KUKA KRL program: MyProgram_032().src

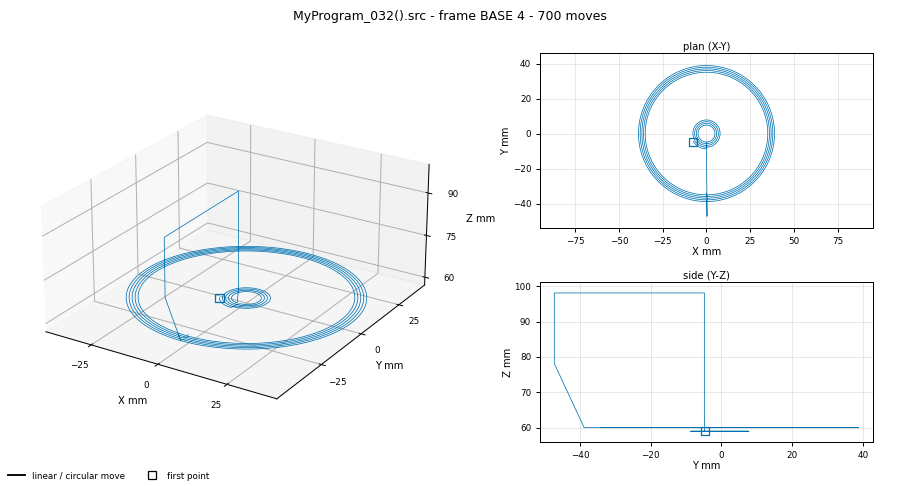
[picture p0: tool path of MyProgram_032().src in frame BASE 4, 700 of 700 moves have a stored position in this frame; points joined in program order, loops and branches not executed]
&ACCESS RVP
&REL 1
&PARAM TEMPLATE = C:\KRC\Roboter\Template\vorgabe
&PARAM EDITMASK = *
DEF MyProgram_032()
; ---- Setting reference (Base) ----
$BASE = BASE_DATA[4]

; --------------------------
; ---- Setting tool (TCP) ----
$TOOL = TOOL_DATA[3]
; --------------------------

$VEL.CP = VEL_APROX_PRINT
Startdeposition()
$VEL.CP = VEL_PRINT
LIN {X -7.455,Y -4.6001,Z 59,A -2.6784,B 0.0017,C -0.0013,E1 0.1616,E2 -630.3527} C_DIS
LIN {X -6.8252,Y -5.4917,Z 59,A -2.6167,B 0.0016,C -0.0015,E1 0.1614,E2 -630.4294} C_DIS
LIN {X -6.0357,Y -6.3443,Z 59,A -2.5577,B 0.0014,C -0.0017,E1 0.1613,E2 -630.4962} C_DIS
LIN {X -5.4394,Y -6.8632,Z 59,A -2.5125,B 0.0012,C -0.0017,E1 0.1611,E2 -630.5421} C_DIS
LIN {X -4.4516,Y -7.5448,Z 59,A -2.4498,B 0.001,C -0.0019,E1 0.1609,E2 -630.5983} C_DIS
LIN {X -3.5499,Y -8.0085,Z 59,A -2.3908,B 0.0007,C -0.002,E1 0.1606,E2 -630.6447} C_DIS
LIN {X -2.4797,Y -8.4018,Z 59,A -2.3387,B 0.0005,C -0.0021,E1 0.1604,E2 -630.6751} C_DIS
LIN {X -1.4775,Y -8.6348,Z 59,A -2.2933,B 0.0002,C -0.0021,E1 0.1601,E2 -630.6944} C_DIS
LIN {X -0.6022,Y -8.7394,Z 59,A -2.2586,B 0,C -0.0021,E1 0.1599,E2 -630.702} C_DIS
LIN {X -0.6022,Y -8.7394,Z 59,A -2.2586,B 0,C -0.0021,E1 0.1599,E2 -630.702} C_DIS
Enddeposition()
LIN {X -0.0216,Y -7.7786,Z 59,A -2.2094,B 0,C -0.0021,E1 0.1599,E2 -630.6884} C_DIS
Startdeposition()
$VEL.CP = VEL_PRINT
LIN {X -1.2171,Y -7.6837,Z 59,A -2.2663,B 0.0003,C -0.0021,E1 0.1602,E2 -630.6706} C_DIS
LIN {X -2.1503,Y -7.4764,Z 59,A -2.3206,B 0.0006,C -0.0021,E1 0.1605,E2 -630.641} C_DIS
LIN {X -3.7783,Y -6.8003,Z 59,A -2.4144,B 0.001,C -0.0019,E1 0.1609,E2 -630.5769} C_DIS
LIN {X -4.6899,Y -6.2006,Z 59,A -2.4825,B 0.0013,C -0.0017,E1 0.1611,E2 -630.5161} C_DIS
LIN {X -5.3546,Y -5.6349,Z 59,A -2.5373,B 0.0014,C -0.0016,E1 0.1613,E2 -630.4612} C_DIS
LIN {X -5.9536,Y -5,Z 59,A -2.5956,B 0.0016,C -0.0014,E1 0.1615,E2 -630.3975} C_DIS
LIN {X -6.5989,Y -4.12,Z 59,A -2.6888,B 0.0018,C -0.0011,E1 0.1617,E2 -630.2903} C_DIS
LIN {X -7.3187,Y -2.6373,Z 59,A -2.7822,B 0.002,C -0.0007,E1 0.1618,E2 -630.1603} C_DIS
LIN {X -7.6546,Y -1.3881,Z 59,A -2.8749,B 0.002,C -0.0004,E1 0.1618,E2 -630.0272} C_DIS
LIN {X -7.776,Y -0.1143,Z 59,A -2.9313,B 0.0021,C -0.0001,E1 0.1619,E2 -629.9218} C_DIS
LIN {X -7.7529,Y 0.5778,Z 59,A -2.9623,B 0.0021,C 0.0001,E1 0.1619,E2 -629.8608} C_DIS
LIN {X -7.6134,Y 1.5989,Z 59,A -3.0373,B 0.0021,C 0.0004,E1 0.1619,E2 -629.7382} C_DIS
LIN {X -7.182,Y 2.9893,Z 59,A -3.0725,B 0.002,C 0.0007,E1 0.1617,E2 -629.6289} C_DIS
LIN {X -6.5899,Y 4.1344,Z 59,A -3.1322,B 0.0018,C 0.0011,E1 0.1615,E2 -629.4997} C_DIS
LIN {X -6.0536,Y 4.8858,Z 59,A -3.1439,B 0.0017,C 0.0013,E1 0.1615,E2 -629.4369} C_DIS
LIN {X -5.0383,Y 5.9273,Z 59,A -3.1697,B 0.0014,C 0.0016,E1 0.1611,E2 -629.33} C_DIS
LIN {X -3.9915,Y 6.6767,Z 59,A -3.1626,B 0.0011,C 0.0018,E1 0.1608,E2 -629.2669} C_DIS
LIN {X -2.8807,Y 7.2264,Z 59,A -3.1481,B 0.0008,C 0.002,E1 0.1605,E2 -629.2169} C_DIS
LIN {X -1.6718,Y 7.5977,Z 59,A -3.1225,B 0.0005,C 0.002,E1 0.1602,E2 -629.1818} C_DIS
LIN {X -0.6433,Y 7.7528,Z 59,A -3.0902,B 0.0002,C 0.0021,E1 0.1599,E2 -629.1689} C_DIS
LIN {X 0.9444,Y 7.7216,Z 59,A -3.0256,B -0.0002,C 0.0021,E1 0.1595,E2 -629.1752} C_DIS
LIN {X 2.2096,Y 7.459,Z 59,A -2.957,B -0.0006,C 0.0021,E1 0.1591,E2 -629.2072} C_DIS
LIN {X 3.4801,Y 6.9537,Z 59,A -2.8858,B -0.0009,C 0.0019,E1 0.1588,E2 -629.252} C_DIS
LIN {X 4.4404,Y 6.3877,Z 59,A -2.8119,B -0.0012,C 0.0018,E1 0.1585,E2 -629.3137} C_DIS
LIN {X 5.2866,Y 5.7073,Z 59,A -2.7397,B -0.0014,C 0.0016,E1 0.1583,E2 -629.383} C_DIS
LIN {X 5.9076,Y 5.0617,Z 59,A -2.6753,B -0.0016,C 0.0014,E1 0.1581,E2 -629.4517} C_DIS
LIN {X 6.6081,Y 4.0967,Z 59,A -2.6072,B -0.0018,C 0.0012,E1 0.158,E2 -629.5347} C_DIS
LIN {X 7.1268,Y 3.1189,Z 59,A -2.5195,B -0.0019,C 0.0009,E1 0.1578,E2 -629.6451} C_DIS
LIN {X 7.5026,Y 2.0563,Z 59,A -2.447,B -0.002,C 0.0006,E1 0.1578,E2 -629.7493} C_DIS
LIN {X 7.7182,Y 0.9735,Z 59,A -2.379,B -0.0021,C 0.0003,E1 0.1577,E2 -629.8562} C_DIS
LIN {X 7.7784,Y -0.1132,Z 59,A -2.3267,B -0.0021,C 0,E1 0.1577,E2 -629.9534} C_DIS
LIN {X 7.718,Y -0.975,Z 59,A -2.2718,B -0.0021,C -0.0003,E1 0.1577,E2 -630.0481} C_DIS
LIN {X 7.4723,Y -2.1625,Z 59,A -2.2174,B -0.0021,C -0.0006,E1 0.1577,E2 -630.1632} C_DIS
LIN {X 7.0963,Y -3.1869,Z 59,A -2.1625,B -0.0019,C -0.0009,E1 0.1579,E2 -630.2768} C_DIS
LIN {X 6.4564,Y -4.34,Z 59,A -2.1405,B -0.0018,C -0.0012,E1 0.1581,E2 -630.3726} C_DIS
LIN {X 5.8227,Y -5.1593,Z 59,A -2.1122,B -0.0016,C -0.0014,E1 0.1583,E2 -630.46} C_DIS
LIN {X 4.8338,Y -6.0906,Z 59,A -2.1217,B -0.0014,C -0.0016,E1 0.1585,E2 -630.5272} C_DIS
LIN {X 4.1033,Y -6.6094,Z 59,A -2.1037,B -0.0011,C -0.0018,E1 0.1588,E2 -630.5947} C_DIS
LIN {X 2.9496,Y -7.1984,Z 59,A -2.1231,B -0.0008,C -0.002,E1 0.1591,E2 -630.6429} C_DIS
LIN {X 1.9713,Y -7.5228,Z 59,A -2.1467,B -0.0006,C -0.002,E1 0.1593,E2 -630.669} C_DIS
LIN {X 0.9282,Y -7.7238,Z 59,A -2.1762,B -0.0003,C -0.0021,E1 0.1596,E2 -630.686} C_DIS
LIN {X -0.0216,Y -7.7786,Z 59,A -2.211,B -0.0001,C -0.0021,E1 0.1598,E2 -630.6879} C_DIS
Enddeposition()
LIN {X -0.0216,Y -7.7786,Z 59,A -2.211,B -0.0001,C -0.0021,E1 0.1598,E2 -630.6879} C_DIS
Startdeposition()
$VEL.CP = VEL_PRINT
LIN {X 0.4638,Y -6.7829,Z 59,A -2.1444,B -0.0003,C -0.0021,E1 0.1596,E2 -630.6937} C_DIS
LIN {X 1.5189,Y -6.6225,Z 59,A -2.1186,B -0.0006,C -0.0021,E1 0.1593,E2 -630.6743} C_DIS
LIN {X 2.5941,Y -6.2842,Z 59,A -2.1115,B -0.001,C -0.0019,E1 0.1589,E2 -630.6275} C_DIS
LIN {X 3.6007,Y -5.7669,Z 59,A -2.1065,B -0.0012,C -0.0017,E1 0.1586,E2 -630.5733} C_DIS
LIN {X 4.2821,Y -5.2763,Z 59,A -2.1172,B -0.0015,C -0.0016,E1 0.1584,E2 -630.5163} C_DIS
LIN {X 4.782,Y -4.8275,Z 59,A -2.1309,B -0.0016,C -0.0014,E1 0.1582,E2 -630.4646} C_DIS
LIN {X 5.2345,Y -4.3312,Z 59,A -2.1517,B -0.0017,C -0.0013,E1 0.1582,E2 -630.4056} C_DIS
LIN {X 5.6368,Y -3.7934,Z 59,A -2.1713,B -0.0018,C -0.0011,E1 0.158,E2 -630.3477} C_DIS
LIN {X 6.1434,Y -2.9119,Z 59,A -2.2267,B -0.002,C -0.0008,E1 0.1578,E2 -630.235} C_DIS
LIN {X 6.5283,Y -1.8963,Z 59,A -2.2993,B -0.0021,C -0.0004,E1 0.1578,E2 -630.1039} C_DIS
LIN {X 6.7263,Y -0.9894,Z 59,A -2.3517,B -0.0021,C -0.0001,E1 0.1577,E2 -630.0047} C_DIS
LIN {X 6.7979,Y 0.0046,Z 59,A -2.4138,B -0.0021,C 0.0002,E1 0.1577,E2 -629.8968} C_DIS
LIN {X 6.6999,Y 1.1554,Z 59,A -2.505,B -0.0021,C 0.0006,E1 0.1577,E2 -629.7594} C_DIS
LIN {X 6.388,Y 2.3182,Z 59,A -2.5672,B -0.002,C 0.0008,E1 0.1577,E2 -629.6587} C_DIS
LIN {X 6.0782,Y 3.0395,Z 59,A -2.6412,B -0.0019,C 0.0011,E1 0.1579,E2 -629.5652} C_DIS
LIN {X 5.6147,Y 3.8293,Z 59,A -2.7146,B -0.0017,C 0.0013,E1 0.1581,E2 -629.4754} C_DIS
LIN {X 5.0506,Y 4.5508,Z 59,A -2.779,B -0.0015,C 0.0015,E1 0.1582,E2 -629.4013} C_DIS
LIN {X 4.3929,Y 5.1881,Z 59,A -2.8476,B -0.0013,C 0.0017,E1 0.1584,E2 -629.3303} C_DIS
LIN {X 3.7651,Y 5.6595,Z 59,A -2.9088,B -0.0011,C 0.0019,E1 0.1587,E2 -629.2727} C_DIS
LIN {X 2.8512,Y 6.1694,Z 59,A -2.975,B -0.0008,C 0.002,E1 0.1589,E2 -629.2192} C_DIS
LIN {X 1.9496,Y 6.5129,Z 59,A -3.0293,B -0.0005,C 0.002,E1 0.1592,E2 -629.1844} C_DIS
LIN {X 0.9311,Y 6.7347,Z 59,A -3.0816,B -0.0001,C 0.0021,E1 0.1596,E2 -629.161} C_DIS
LIN {X -0.1024,Y 6.7978,Z 59,A -3.1177,B 0.0002,C 0.0021,E1 0.1599,E2 -629.1611} C_DIS
LIN {X -1.1045,Y 6.7084,Z 59,A -3.1431,B 0.0005,C 0.0021,E1 0.1602,E2 -629.177} C_DIS
LIN {X -1.8211,Y 6.5455,Z 59,A -3.1548,B 0.0008,C 0.0021,E1 0.1605,E2 -629.199} C_DIS
LIN {X -2.7429,Y 6.2156,Z 59,A -3.1609,B 0.001,C 0.0019,E1 0.1607,E2 -629.2412} C_DIS
LIN {X -3.608,Y 5.7571,Z 59,A -3.1711,B 0.0012,C 0.0018,E1 0.1609,E2 -629.2824} C_DIS
LIN {X -4.2239,Y 5.3274,Z 59,A -3.143,B 0.0015,C 0.0015,E1 0.1612,E2 -629.3512} C_DIS
LIN {X -4.9859,Y 4.6149,Z 59,A -3.1236,B 0.0017,C 0.0013,E1 0.1614,E2 -629.4286} C_DIS
LIN {X -5.6898,Y 3.7213,Z 59,A -3.0827,B 0.0019,C 0.001,E1 0.1616,E2 -629.5328} C_DIS
LIN {X -6.1512,Y 2.895,Z 59,A -3.0358,B 0.002,C 0.0007,E1 0.1618,E2 -629.6311} C_DIS
LIN {X -6.4104,Y 2.2507,Z 59,A -3.0263,B 0.002,C 0.0007,E1 0.1618,E2 -629.6772} C_DIS
LIN {X -6.6245,Y 1.5285,Z 59,A -2.9621,B 0.0021,C 0.0003,E1 0.1618,E2 -629.7793} C_DIS
LIN {X -6.7591,Y 0.6788,Z 59,A -2.9085,B 0.0021,C 0.0001,E1 0.1619,E2 -629.8734} C_DIS
LIN {X -6.7963,Y -0.1808,Z 59,A -2.8206,B 0.0021,C -0.0003,E1 0.1619,E2 -629.9985} C_DIS
LIN {X -6.5543,Y -1.8059,Z 59,A -2.7336,B 0.0021,C -0.0007,E1 0.1619,E2 -630.1452} C_DIS
LIN {X -6.2054,Y -2.7775,Z 59,A -2.6265,B 0.0019,C -0.0011,E1 0.1617,E2 -630.2806} C_DIS
LIN {X -5.4796,Y -4.0189,Z 59,A -2.5356,B 0.0016,C -0.0014,E1 0.1615,E2 -630.3978} C_DIS
LIN {X -4.7369,Y -4.8769,Z 59,A -2.4497,B 0.0014,C -0.0016,E1 0.1612,E2 -630.4935} C_DIS
LIN {X -4.0591,Y -5.4541,Z 59,A -2.385,B 0.0011,C -0.0018,E1 0.161,E2 -630.5584} C_DIS
LIN {X -3.0573,Y -6.0679,Z 59,A -2.3109,B 0.0008,C -0.002,E1 0.1607,E2 -630.6226} C_DIS
LIN {X -2.2512,Y -6.4098,Z 59,A -2.2612,B 0.0006,C -0.002,E1 0.1605,E2 -630.6579} C_DIS
LIN {X -1.4085,Y -6.6473,Z 59,A -2.2158,B 0.0003,C -0.0021,E1 0.1602,E2 -630.683} C_DIS
LIN {X -0.2496,Y -6.7939,Z 59,A -2.1672,B 0,C -0.0021,E1 0.1598,E2 -630.6961} C_DIS
LIN {X -0.2496,Y -6.7939,Z 59,A -2.1672,B 0,C -0.0021,E1 0.1598,E2 -630.6961} C_DIS
Enddeposition()
LIN {X -0.0178,Y -5.8179,Z 59,A -2.1057,B 0,C -0.0021,E1 0.1598,E2 -630.7068} C_DIS
Startdeposition()
$VEL.CP = VEL_PRINT
LIN {X -0.946,Y -5.7346,Z 59,A -2.153,B 0.0003,C -0.0021,E1 0.1602,E2 -630.6896} C_DIS
LIN {X -1.6727,Y -5.5675,Z 59,A -2.1975,B 0.0006,C -0.0021,E1 0.1605,E2 -630.6641} C_DIS
LIN {X -2.7269,Y -5.1392,Z 59,A -2.2839,B 0.001,C -0.0019,E1 0.1609,E2 -630.5974} C_DIS
LIN {X -3.5542,Y -4.5969,Z 59,A -2.3648,B 0.0013,C -0.0017,E1 0.1612,E2 -630.5231} C_DIS
LIN {X -4.1461,Y -4.072,Z 59,A -2.4337,B 0.0015,C -0.0015,E1 0.1614,E2 -630.4532} C_DIS
LIN {X -4.6623,Y -3.4725,Z 59,A -2.5154,B 0.0017,C -0.0013,E1 0.1616,E2 -630.3647} C_DIS
LIN {X -5.0883,Y -2.8057,Z 59,A -2.5873,B 0.0019,C -0.0011,E1 0.1617,E2 -630.28} C_DIS
LIN {X -5.4237,Y -2.0891,Z 59,A -2.6666,B 0.002,C -0.0008,E1 0.1618,E2 -630.1825} C_DIS
LIN {X -5.7408,Y -0.9445,Z 59,A -2.7856,B 0.0021,C -0.0004,E1 0.1619,E2 -630.0268} C_DIS
LIN {X -5.8118,Y 0.0093,Z 59,A -2.8735,B 0.0021,C 0,E1 0.1619,E2 -629.9014} C_DIS
LIN {X -5.759,Y 0.7724,Z 59,A -2.938,B 0.0021,C 0.0002,E1 0.1619,E2 -629.8031} C_DIS
LIN {X -5.6094,Y 1.5226,Z 59,A -2.9999,B 0.0021,C 0.0005,E1 0.1619,E2 -629.7042} C_DIS
LIN {X -5.3597,Y 2.2456,Z 59,A -3.0547,B 0.0021,C 0.0008,E1 0.1618,E2 -629.61} C_DIS
LIN {X -5.019,Y 2.9305,Z 59,A -3.1032,B 0.0019,C 0.0011,E1 0.1616,E2 -629.5204} C_DIS
LIN {X -4.5915,Y 3.565,Z 59,A -3.1429,B 0.0017,C 0.0013,E1 0.1615,E2 -629.4384} C_DIS
LIN {X -3.8274,Y 4.3817,Z 59,A -3.1905,B 0.0015,C 0.0016,E1 0.1612,E2 -629.3284} C_DIS
LIN {X -3.012,Y 4.9721,Z 59,A -3.2116,B 0.0012,C 0.0018,E1 0.1609,E2 -629.2524} C_DIS
LIN {X -2.2952,Y 5.3395,Z 59,A -3.2138,B 0.0009,C 0.002,E1 0.1606,E2 -629.2081} C_DIS
LIN {X -1.1834,Y 5.6963,Z 59,A -3.2008,B 0.0005,C 0.0021,E1 0.1602,E2 -629.1645} C_DIS
LIN {X -0.5624,Y 5.789,Z 59,A -3.1855,B 0.0003,C 0.0021,E1 0.16,E2 -629.1526} C_DIS
LIN {X 0.5083,Y 5.7955,Z 59,A -3.1402,B -0.0002,C 0.0021,E1 0.1595,E2 -629.1574} C_DIS
LIN {X 1.8592,Y 5.5064,Z 59,A -3.0638,B -0.0007,C 0.0021,E1 0.159,E2 -629.1951} C_DIS
LIN {X 2.536,Y 5.2283,Z 59,A -3.0134,B -0.0009,C 0.002,E1 0.1588,E2 -629.2318} C_DIS
LIN {X 3.1747,Y 4.8709,Z 59,A -2.9526,B -0.0012,C 0.0018,E1 0.1586,E2 -629.2837} C_DIS
LIN {X 3.7611,Y 4.4328,Z 59,A -2.888,B -0.0014,C 0.0017,E1 0.1583,E2 -629.3448} C_DIS
LIN {X 4.2878,Y 3.9244,Z 59,A -2.8191,B -0.0016,C 0.0015,E1 0.1581,E2 -629.4156} C_DIS
LIN {X 4.7461,Y 3.3538,Z 59,A -2.7512,B -0.0017,C 0.0013,E1 0.158,E2 -629.4908} C_DIS
LIN {X 5.1315,Y 2.7317,Z 59,A -2.6748,B -0.0019,C 0.001,E1 0.1578,E2 -629.5794} C_DIS
LIN {X 5.4342,Y 2.0652,Z 59,A -2.6031,B -0.002,C 0.0008,E1 0.1578,E2 -629.6684} C_DIS
LIN {X 5.7407,Y 0.9435,Z 59,A -2.4808,B -0.0021,C 0.0004,E1 0.1576,E2 -629.8277} C_DIS
LIN {X 5.8175,Y 0.018,Z 59,A -2.3792,B -0.0021,C 0,E1 0.1576,E2 -629.9666} C_DIS
LIN {X 5.6764,Y -1.2466,Z 59,A -2.283,B -0.0021,C -0.0005,E1 0.1576,E2 -630.123} C_DIS
LIN {X 5.4306,Y -2.0706,Z 59,A -2.2172,B -0.0021,C -0.0008,E1 0.1578,E2 -630.2338} C_DIS
LIN {X 4.816,Y -3.2633,Z 59,A -2.1283,B -0.0018,C -0.0012,E1 0.1581,E2 -630.3974} C_DIS
LIN {X 4.2399,Y -3.9837,Z 59,A -2.0854,B -0.0016,C -0.0015,E1 0.1583,E2 -630.493} C_DIS
LIN {X 3.4525,Y -4.6828,Z 59,A -2.0587,B -0.0013,C -0.0018,E1 0.1586,E2 -630.579} C_DIS
LIN {X 2.5057,Y -5.2504,Z 59,A -2.0587,B -0.001,C -0.0019,E1 0.1589,E2 -630.6383} C_DIS
LIN {X 1.6471,Y -5.5797,Z 59,A -2.0641,B -0.0007,C -0.0021,E1 0.1592,E2 -630.6783} C_DIS
LIN {X 0.8082,Y -5.7613,Z 59,A -2.0803,B -0.0004,C -0.0021,E1 0.1595,E2 -630.7005} C_DIS
LIN {X -0.0178,Y -5.8179,Z 59,A -2.1067,B -0.0001,C -0.0021,E1 0.1597,E2 -630.7065} C_DIS
Enddeposition()
LIN {X -0.0178,Y -5.8179,Z 59,A -2.1067,B -0.0001,C -0.0021,E1 0.1597,E2 -630.7065} C_DIS
Startdeposition()
$VEL.CP = VEL_PRINT
LIN {X 0.4835,Y -4.8072,Z 59,A -2.0593,B -0.0004,C -0.0021,E1 0.1595,E2 -630.6919} C_DIS
LIN {X 1.1408,Y -4.6961,Z 59,A -2.0523,B -0.0007,C -0.0021,E1 0.1592,E2 -630.6701} C_DIS
LIN {X 1.7761,Y -4.4937,Z 59,A -2.0556,B -0.0009,C -0.0019,E1 0.1589,E2 -630.6349} C_DIS
LIN {X 2.3773,Y -4.2055,Z 59,A -2.0664,B -0.0012,C -0.0018,E1 0.1587,E2 -630.5896} C_DIS
LIN {X 2.9348,Y -3.8398,Z 59,A -2.0962,B -0.0014,C -0.0016,E1 0.1584,E2 -630.5234} C_DIS
LIN {X 3.4338,Y -3.3976,Z 59,A -2.1258,B -0.0016,C -0.0014,E1 0.1582,E2 -630.4562} C_DIS
LIN {X 3.8697,Y -2.8933,Z 59,A -2.1739,B -0.0018,C -0.0012,E1 0.158,E2 -630.3701} C_DIS
LIN {X 4.2319,Y -2.3335,Z 59,A -2.2266,B -0.0019,C -0.0009,E1 0.1579,E2 -630.2796} C_DIS
LIN {X 4.5124,Y -1.7287,Z 59,A -2.2933,B -0.0021,C -0.0006,E1 0.1578,E2 -630.1762} C_DIS
LIN {X 4.7068,Y -1.0908,Z 59,A -2.3557,B -0.0021,C -0.0003,E1 0.1577,E2 -630.0788} C_DIS
LIN {X 4.8134,Y -0.4327,Z 59,A -2.4333,B -0.0021,C 0,E1 0.1577,E2 -629.9686} C_DIS
LIN {X 4.8257,Y 0.234,Z 59,A -2.5121,B -0.0021,C 0.0003,E1 0.1577,E2 -629.8604} C_DIS
LIN {X 4.7472,Y 0.8961,Z 59,A -2.5877,B -0.0021,C 0.0006,E1 0.1577,E2 -629.7592} C_DIS
LIN {X 4.5804,Y 1.5415,Z 59,A -2.6704,B -0.002,C 0.0008,E1 0.1577,E2 -629.6548} C_DIS
LIN {X 4.3256,Y 2.1577,Z 59,A -2.7524,B -0.0018,C 0.0011,E1 0.1579,E2 -629.5559} C_DIS
LIN {X 3.9864,Y 2.7319,Z 59,A -2.8351,B -0.0017,C 0.0014,E1 0.1581,E2 -629.4613} C_DIS
LIN {X 3.5709,Y 3.2534,Z 59,A -2.9023,B -0.0015,C 0.0016,E1 0.1583,E2 -629.3874} C_DIS
LIN {X 3.0895,Y 3.7143,Z 59,A -2.9724,B -0.0012,C 0.0018,E1 0.1585,E2 -629.3158} C_DIS
LIN {X 2.5491,Y 4.1049,Z 59,A -3.0375,B -0.001,C 0.0019,E1 0.1587,E2 -629.2545} C_DIS
LIN {X 1.9593,Y 4.4158,Z 59,A -3.0895,B -0.0007,C 0.002,E1 0.159,E2 -629.2115} C_DIS
LIN {X 1.333,Y 4.6442,Z 59,A -3.1351,B -0.0004,C 0.0021,E1 0.1593,E2 -629.1798} C_DIS
LIN {X 0.6812,Y 4.7845,Z 59,A -3.1713,B -0.0001,C 0.0021,E1 0.1596,E2 -629.1623} C_DIS
LIN {X 0.0161,Y 4.8297,Z 59,A -3.1966,B 0.0002,C 0.0021,E1 0.1599,E2 -629.16} C_DIS
LIN {X -0.6492,Y 4.7883,Z 59,A -3.2102,B 0.0005,C 0.0021,E1 0.1602,E2 -629.1732} C_DIS
LIN {X -1.3018,Y 4.6517,Z 59,A -3.2164,B 0.0007,C 0.0021,E1 0.1604,E2 -629.197} C_DIS
LIN {X -1.9305,Y 4.43,Z 59,A -3.2059,B 0.001,C 0.0019,E1 0.1607,E2 -629.2404} C_DIS
LIN {X -2.5216,Y 4.1215,Z 59,A -3.1897,B 0.0013,C 0.0017,E1 0.161,E2 -629.2914} C_DIS
LIN {X -3.0655,Y 3.7359,Z 59,A -3.1613,B 0.0015,C 0.0015,E1 0.1612,E2 -629.3562} C_DIS
LIN {X -3.5515,Y 3.2793,Z 59,A -3.1218,B 0.0017,C 0.0013,E1 0.1614,E2 -629.4327} C_DIS
LIN {X -3.9683,Y 2.7587,Z 59,A -3.0712,B 0.0019,C 0.0011,E1 0.1616,E2 -629.5205} C_DIS
LIN {X -4.3091,Y 2.1856,Z 59,A -3.0206,B 0.0019,C 0.0008,E1 0.1617,E2 -629.6076} C_DIS
LIN {X -4.57,Y 1.5719,Z 59,A -2.9567,B 0.0021,C 0.0005,E1 0.1618,E2 -629.7067} C_DIS
LIN {X -4.7428,Y 0.9279,Z 59,A -2.8853,B 0.0021,C 0.0002,E1 0.1619,E2 -629.8115} C_DIS
LIN {X -4.8246,Y 0.2661,Z 59,A -2.8155,B 0.0021,C -0.0001,E1 0.1619,E2 -629.912} C_DIS
LIN {X -4.8165,Y -0.4006,Z 59,A -2.7377,B 0.0021,C -0.0004,E1 0.1619,E2 -630.0175} C_DIS
LIN {X -4.7162,Y -1.0599,Z 59,A -2.6572,B 0.0021,C -0.0006,E1 0.1619,E2 -630.1221} C_DIS
LIN {X -4.5245,Y -1.6986,Z 59,A -2.5778,B 0.0019,C -0.0009,E1 0.1618,E2 -630.2215} C_DIS
LIN {X -4.247,Y -2.3049,Z 59,A -2.4993,B 0.0018,C -0.0012,E1 0.1616,E2 -630.3156} C_DIS
LIN {X -3.8891,Y -2.8676,Z 59,A -2.4258,B 0.0016,C -0.0014,E1 0.1615,E2 -630.4} C_DIS
LIN {X -3.4582,Y -3.3764,Z 59,A -2.3529,B 0.0014,C -0.0016,E1 0.1613,E2 -630.479} C_DIS
LIN {X -2.9611,Y -3.821,Z 59,A -2.2854,B 0.0012,C -0.0018,E1 0.1611,E2 -630.5475} C_DIS
LIN {X -2.4067,Y -4.1916,Z 59,A -2.2248,B 0.0009,C -0.0019,E1 0.1608,E2 -630.6039} C_DIS
LIN {X -1.806,Y -4.4809,Z 59,A -2.1713,B 0.0007,C -0.002,E1 0.1605,E2 -630.6482} C_DIS
LIN {X -1.1721,Y -4.6877,Z 59,A -2.1276,B 0.0004,C -0.0021,E1 0.1602,E2 -630.6777} C_DIS
LIN {X -0.5156,Y -4.8034,Z 59,A -2.0926,B 0.0001,C -0.0021,E1 0.16,E2 -630.694} C_DIS
LIN {X -0.5156,Y -4.8034,Z 59,A -2.0926,B 0.0001,C -0.0021,E1 0.16,E2 -630.694} C_DIS
Enddeposition()
LIN {X -0.0162,Y -4.8336,Z 64,A -2.0645,B 0.0001,C -0.0021,E1 0.1599,E2 -630.6953} C_DIS
LIN {X -0.0162,Y -4.8331,Z 79,A -2.0395,B 0.0001,C -0.0021,E1 0.1599,E2 -630.6941} C_DIS
LIN {X -0.0162,Y -4.8331,Z 98.1262,A -2.0155,B 0.0001,C -0.0021,E1 0.1599,E2 -630.6939} C_DIS
LIN {X 0.3094,Y -47.296,Z 98.1262,A -95.6566,B 24.8514,C -2.8125,E1 25.0031,E2 -541.3733} C_DIS
LIN {X 0.3094,Y -47.296,Z 78.1262,A -95.326,B 24.8658,C -2.6735,E1 25.0031,E2 -541.3733} C_DIS
LIN {X 0.1976,Y -40.9577,Z 64.5315,A -95.3613,B 24.8643,C -2.6884,E1 25.0031,E2 -541.3733} C_DIS
LIN {X 0.1603,Y -38.845,Z 60,A -95.3746,B 24.8637,C -2.694,E1 25.0031,E2 -541.3733} C_DIS
Startdeposition()
$VEL.CP = VEL_PRINT
LIN {X 2.5506,Y -38.7626,Z 60,A -91.6975,B 24.8634,C -2.6973,E1 25.0134,E2 -545.0572} C_DIS
LIN {X 4.8829,Y -38.5385,Z 60,A -88.2483,B 24.8632,C -2.6992,E1 25.023,E2 -548.5085} C_DIS
LIN {X 7.1105,Y -38.1904,Z 60,A -84.9063,B 24.8629,C -2.702,E1 25.0322,E2 -551.8535} C_DIS
LIN {X 9.4388,Y -37.682,Z 60,A -81.4521,B 24.8626,C -2.7044,E1 25.0416,E2 -555.3086} C_DIS
LIN {X 11.7431,Y -37.0285,Z 60,A -78.1432,B 24.8626,C -2.7051,E1 25.0504,E2 -558.6134} C_DIS
LIN {X 13.7916,Y -36.3158,Z 60,A -74.7707,B 24.8619,C -2.7118,E1 25.0593,E2 -561.9946} C_DIS
LIN {X 15.7532,Y -35.5091,Z 60,A -71.6406,B 24.8614,C -2.7163,E1 25.0673,E2 -565.128} C_DIS
LIN {X 17.8421,Y -34.507,Z 60,A -68.2076,B 24.8608,C -2.722,E1 25.0759,E2 -568.5653} C_DIS
LIN {X 19.9714,Y -33.3203,Z 60,A -64.5882,B 24.8602,C -2.7288,E1 25.0847,E2 -572.1897} C_DIS
LIN {X 21.9767,Y -32.0324,Z 60,A -61.1679,B 24.8596,C -2.7341,E1 25.0926,E2 -575.6112} C_DIS
LIN {X 23.9094,Y -30.6176,Z 60,A -57.5746,B 24.8588,C -2.7423,E1 25.1006,E2 -579.211} C_DIS
LIN {X 25.799,Y -29.0427,Z 60,A -53.9773,B 24.858,C -2.7499,E1 25.1083,E2 -582.8122} C_DIS
LIN {X 27.4922,Y -27.4456,Z 60,A -50.5627,B 24.8572,C -2.7576,E1 25.1151,E2 -586.2309} C_DIS
LIN {X 29.1013,Y -25.7325,Z 60,A -47.1744,B 24.8564,C -2.765,E1 25.1215,E2 -589.6215} C_DIS
LIN {X 30.6273,Y -23.897,Z 60,A -43.5888,B 24.8553,C -2.7751,E1 25.1277,E2 -593.2144} C_DIS
LIN {X 32.0997,Y -21.8785,Z 60,A -39.9683,B 24.8544,C -2.7839,E1 25.1336,E2 -596.8382} C_DIS
LIN {X 33.4319,Y -19.7826,Z 60,A -36.3645,B 24.8534,C -2.7932,E1 25.1388,E2 -600.4456} C_DIS
LIN {X 34.5386,Y -17.7803,Z 60,A -32.939,B 24.8523,C -2.8037,E1 25.1433,E2 -603.878} C_DIS
LIN {X 35.585,Y -15.5806,Z 60,A -29.592,B 24.8516,C -2.8103,E1 25.1472,E2 -607.2222} C_DIS
LIN {X 36.4119,Y -13.5347,Z 60,A -26.2439,B 24.8504,C -2.8215,E1 25.1506,E2 -610.5785} C_DIS
LIN {X 37.1968,Y -11.2013,Z 60,A -22.6698,B 24.8494,C -2.8317,E1 25.1537,E2 -614.1563} C_DIS
LIN {X 37.7978,Y -8.9641,Z 60,A -19.2995,B 24.8483,C -2.8415,E1 25.156,E2 -617.5303} C_DIS
LIN {X 38.2751,Y -6.6414,Z 60,A -15.8959,B 24.8473,C -2.8508,E1 25.1578,E2 -620.9361} C_DIS
LIN {X 38.5923,Y -4.4369,Z 60,A -12.5033,B 24.846,C -2.8629,E1 25.159,E2 -624.3373} C_DIS
LIN {X 38.789,Y -2.1119,Z 60,A -9.0204,B 24.8448,C -2.8744,E1 25.1597,E2 -627.8267} C_DIS
LIN {X 38.8442,Y -0.4767,Z 60,A -6.8142,B 24.8443,C -2.8785,E1 25.1597,E2 -630.0295} C_DIS
LIN {X 38.8078,Y 1.7318,Z 60,A -3.3527,B 24.8428,C -2.892,E1 25.1595,E2 -633.5025} C_DIS
LIN {X 38.6469,Y 3.9339,Z 60,A -0.3536,B 24.8422,C -2.8979,E1 25.1587,E2 -636.4977} C_DIS
LIN {X 38.3557,Y 6.1594,Z 60,A 2.9747,B 24.8411,C -2.9084,E1 25.1574,E2 -639.8312} C_DIS
LIN {X 37.9352,Y 8.3648,Z 60,A 6.3462,B 24.8399,C -2.9194,E1 25.1555,E2 -643.209} C_DIS
LIN {X 37.3638,Y 10.6297,Z 60,A 9.814,B 24.8387,C -2.93,E1 25.153,E2 -646.682} C_DIS
LIN {X 36.7294,Y 12.6484,Z 60,A 12.9236,B 24.8377,C -2.9388,E1 25.1503,E2 -649.795} C_DIS
LIN {X 35.8848,Y 14.8769,Z 60,A 16.2289,B 24.837,C -2.9454,E1 25.1469,E2 -653.0975} C_DIS
LIN {X 35.1119,Y 16.6199,Z 60,A 19.0029,B 24.8362,C -2.9526,E1 25.1436,E2 -655.8735} C_DIS
LIN {X 34.1463,Y 18.5222,Z 60,A 22.3064,B 24.835,C -2.9635,E1 25.1393,E2 -659.1854} C_DIS
LIN {X 32.9162,Y 20.6293,Z 60,A 25.8645,B 24.834,C -2.9721,E1 25.1342,E2 -662.7458} C_DIS
LIN {X 31.6722,Y 22.4927,Z 60,A 29.2129,B 24.833,C -2.9809,E1 25.1289,E2 -666.0986} C_DIS
LIN {X 30.2957,Y 24.3156,Z 60,A 32.6004,B 24.8321,C -2.9891,E1 25.1231,E2 -669.4895} C_DIS
LIN {X 28.6843,Y 26.1967,Z 60,A 36.2049,B 24.8312,C -2.9964,E1 25.1164,E2 -673.0952} C_DIS
LIN {X 27.0874,Y 27.8451,Z 60,A 39.6045,B 24.8304,C -3.0036,E1 25.1097,E2 -676.4976} C_DIS
LIN {X 25.2558,Y 29.5161,Z 60,A 43.2116,B 24.8297,C -3.0099,E1 25.1021,E2 -680.1052} C_DIS
LIN {X 23.474,Y 30.9524,Z 60,A 46.6037,B 24.829,C -3.0161,E1 25.0946,E2 -683.4996} C_DIS
LIN {X 21.465,Y 32.3776,Z 60,A 50.1931,B 24.8284,C -3.0213,E1 25.0864,E2 -687.089} C_DIS
LIN {X 19.5416,Y 33.574,Z 60,A 53.5368,B 24.8279,C -3.0261,E1 25.0784,E2 -690.4339} C_DIS
LIN {X 17.405,Y 34.7295,Z 60,A 57.071,B 24.8274,C -3.03,E1 25.0696,E2 -693.9673} C_DIS
LIN {X 15.305,Y 35.704,Z 60,A 60.3841,B 24.8272,C -3.0323,E1 25.0612,E2 -697.2778} C_DIS
LIN {X 13.4006,Y 36.462,Z 60,A 63.3814,B 24.8269,C -3.0347,E1 25.0534,E2 -700.2743} C_DIS
LIN {X 11.2013,Y 37.1968,Z 60,A 66.8393,B 24.8265,C -3.0379,E1 25.0442,E2 -703.7333} C_DIS
LIN {X 8.9641,Y 37.7978,Z 60,A 70.2291,B 24.8263,C -3.0395,E1 25.035,E2 -707.1219} C_DIS
LIN {X 6.6414,Y 38.2751,Z 60,A 73.654,B 24.8263,C -3.0399,E1 25.0256,E2 -710.5437} C_DIS
LIN {X 4.4369,Y 38.5923,Z 60,A 77.0695,B 24.826,C -3.0423,E1 25.0161,E2 -713.9623} C_DIS
LIN {X 2.1119,Y 38.789,Z 60,A 80.5771,B 24.826,C -3.0433,E1 25.0064,E2 -717.4705} C_DIS
LIN {X -0.3374,Y 38.8451,Z 60,A 84.0988,B 24.8261,C -3.0415,E1 24.9965,E2 -720.9876} C_DIS
LIN {X -2.6658,Y 38.7549,Z 60,A 87.6028,B 24.8261,C -3.0411,E1 24.9868,E2 -724.4917} C_DIS
LIN {X -4.8829,Y 38.5385,Z 60,A 90.9409,B 24.8263,C -3.0399,E1 24.9775,E2 -727.8292} C_DIS
LIN {X -7.1105,Y 38.1904,Z 60,A 94.2943,B 24.8265,C -3.0379,E1 24.9683,E2 -731.181} C_DIS
LIN {X -9.4388,Y 37.682,Z 60,A 97.7632,B 24.827,C -3.0341,E1 24.9589,E2 -734.6457} C_DIS
LIN {X -11.7431,Y 37.0285,Z 60,A 101.0888,B 24.8277,C -3.0278,E1 24.95,E2 -737.9618} C_DIS
LIN {X -13.7916,Y 36.3158,Z 60,A 104.4811,B 24.8279,C -3.0261,E1 24.9411,E2 -741.3569} C_DIS
LIN {X -15.9378,Y 35.4262,Z 60,A 107.8689,B 24.8285,C -3.0208,E1 24.9324,E2 -744.7399} C_DIS
LIN {X -17.8903,Y 34.4817,Z 60,A 111.1429,B 24.829,C -3.0166,E1 24.9243,E2 -748.0127} C_DIS
LIN {X -19.9714,Y 33.3203,Z 60,A 114.7391,B 24.8295,C -3.0114,E1 24.9156,E2 -751.6072} C_DIS
LIN {X -21.9767,Y 32.0324,Z 60,A 118.1895,B 24.8304,C -3.0041,E1 24.9076,E2 -755.0514} C_DIS
LIN {X -23.9,Y 30.625,Z 60,A 121.8108,B 24.8311,C -2.9981,E1 24.8995,E2 -758.6714} C_DIS
LIN {X -25.799,Y 29.0427,Z 60,A 125.4511,B 24.832,C -2.99,E1 24.8918,E2 -762.3067} C_DIS
LIN {X -27.4922,Y 27.4456,Z 60,A 128.9027,B 24.8328,C -2.9823,E1 24.8849,E2 -765.7542} C_DIS
LIN {X -29.1013,Y 25.7325,Z 60,A 132.3296,B 24.8338,C -2.9734,E1 24.8785,E2 -769.175} C_DIS
LIN {X -30.6273,Y 23.897,Z 60,A 135.958,B 24.8347,C -2.9655,E1 24.8722,E2 -772.8015} C_DIS
LIN {X -32.0997,Y 21.8785,Z 60,A 139.6234,B 24.8358,C -2.9555,E1 24.8663,E2 -776.4609} C_DIS
LIN {X -33.4319,Y 19.7826,Z 60,A 143.2738,B 24.837,C -2.9452,E1 24.8609,E2 -780.1054} C_DIS
LIN {X -34.507,Y 17.8421,Z 60,A 146.4298,B 24.8382,C -2.9347,E1 24.8568,E2 -783.253} C_DIS
LIN {X -35.3611,Y 16.0828,Z 60,A 149.3247,B 24.8391,C -2.9264,E1 24.8534,E2 -786.1437} C_DIS
LIN {X -36.1191,Y 14.2992,Z 60,A 152.1939,B 24.84,C -2.918,E1 24.8503,E2 -789.0089} C_DIS
LIN {X -36.8008,Y 12.4397,Z 60,A 155.3647,B 24.8407,C -2.9117,E1 24.8474,E2 -792.1826} C_DIS
LIN {X -37.4898,Y 10.1765,Z 60,A 158.8663,B 24.8418,C -2.9012,E1 24.8447,E2 -795.6792} C_DIS
LIN {X -38.0322,Y 7.9126,Z 60,A 162.3294,B 24.843,C -2.8908,E1 24.8426,E2 -799.138} C_DIS
LIN {X -38.4265,Y 5.7,Z 60,A 165.6906,B 24.8441,C -2.881,E1 24.8411,E2 -802.4955} C_DIS
LIN {X -38.703,Y 3.3329,Z 60,A 169.1687,B 24.8453,C -2.8696,E1 24.8402,E2 -805.9672} C_DIS
LIN {X -38.8421,Y 0.5894,Z 60,A 172.2889,B 24.8477,C -2.8476,E1 24.8398,E2 -809.0537} C_DIS
LIN {X -38.8201,Y -1.4298,Z 60,A 176.2675,B 24.8476,C -2.8483,E1 24.84,E2 -813.0578} C_DIS
LIN {X -38.6529,Y -3.8759,Z 60,A 179.763,B 24.8489,C -2.8359,E1 24.8408,E2 -816.5446} C_DIS
LIN {X -38.3557,Y -6.1594,Z 60,A -176.8398,B 24.85,C -2.8255,E1 24.8422,E2 -819.9372} C_DIS
LIN {X -37.9352,Y -8.3648,Z 60,A -173.4094,B 24.851,C -2.8167,E1 24.8441,E2 -823.3668} C_DIS
LIN {X -37.3638,Y -10.6297,Z 60,A -169.8969,B 24.852,C -2.8072,E1 24.8466,E2 -826.8769} C_DIS
LIN {X -36.6496,Y -12.8776,Z 60,A -166.4148,B 24.853,C -2.7971,E1 24.8497,E2 -830.3549} C_DIS
LIN {X -35.8848,Y -14.8769,Z 60,A -163.3936,B 24.8541,C -2.7868,E1 24.8528,E2 -833.3682} C_DIS
LIN {X -35.1119,Y -16.6199,Z 60,A -160.584,B 24.8549,C -2.779,E1 24.8561,E2 -836.1745} C_DIS
LIN {X -34.1463,Y -18.5222,Z 60,A -157.2415,B 24.8556,C -2.7727,E1 24.8604,E2 -839.5198} C_DIS
LIN {X -32.9162,Y -20.6293,Z 60,A -153.639,B 24.8566,C -2.7635,E1 24.8656,E2 -843.1188} C_DIS
LIN {X -31.6722,Y -22.4927,Z 60,A -150.2524,B 24.8573,C -2.7563,E1 24.871,E2 -846.5049} C_DIS
LIN {X -30.1885,Y -24.4479,Z 60,A -146.6172,B 24.8582,C -2.748,E1 24.8773,E2 -850.1375} C_DIS
LIN {X -28.6258,Y -26.2604,Z 60,A -143.102,B 24.859,C -2.7401,E1 24.8838,E2 -853.6496} C_DIS
LIN {X -27.0874,Y -27.8451,Z 60,A -139.7547,B 24.8596,C -2.7344,E1 24.8904,E2 -856.9975} C_DIS
LIN {X -25.2558,Y -29.5161,Z 60,A -136.1157,B 24.8603,C -2.7273,E1 24.898,E2 -860.6338} C_DIS
LIN {X -23.474,Y -30.9524,Z 60,A -132.6961,B 24.8609,C -2.7219,E1 24.9055,E2 -864.0531} C_DIS
LIN {X -21.465,Y -32.3776,Z 60,A -129.08,B 24.8615,C -2.7159,E1 24.9139,E2 -867.6671} C_DIS
LIN {X -19.5416,Y -33.574,Z 60,A -125.7143,B 24.8619,C -2.7115,E1 24.9219,E2 -871.0325} C_DIS
LIN {X -17.405,Y -34.7295,Z 60,A -122.247,B 24.8625,C -2.7056,E1 24.9305,E2 -874.4953} C_DIS
LIN {X -15.5806,Y -35.585,Z 60,A -119.3338,B 24.8629,C -2.7017,E1 24.9379,E2 -877.4063} C_DIS
LIN {X -13.5347,Y -36.4119,Z 60,A -115.9553,B 24.8631,C -2.7002,E1 24.9467,E2 -880.7886} C_DIS
LIN {X -11.2013,Y -37.1968,Z 60,A -112.3499,B 24.8634,C -2.6972,E1 24.9563,E2 -884.3932} C_DIS
LIN {X -8.9641,Y -37.7978,Z 60,A -108.9513,B 24.8636,C -2.6951,E1 24.9655,E2 -887.7917} C_DIS
LIN {X -6.6414,Y -38.2751,Z 60,A -105.5203,B 24.8638,C -2.6929,E1 24.9749,E2 -891.2212} C_DIS
LIN {X -4.4369,Y -38.5923,Z 60,A -102.1018,B 24.8637,C -2.6941,E1 24.9844,E2 -894.6451} C_DIS
LIN {X -2.1119,Y -38.789,Z 60,A -98.5942,B 24.8636,C -2.6951,E1 24.9942,E2 -898.1563} C_DIS
LIN {X 0.1603,Y -38.845,Z 60,A -95.3754,B 24.8637,C -2.6939,E1 25.0031,E2 -901.3724} C_DIS
Enddeposition()
LIN {X 0.1603,Y -38.845,Z 60,A -95.3754,B 24.8637,C -2.6939,E1 25.0031,E2 -901.3724} C_DIS
Startdeposition()
$VEL.CP = VEL_PRINT
LIN {X -0.1005,Y -37.8884,Z 60,A -97.4636,B 24.8643,C -2.688,E1 24.9973,E2 -899.2703} C_DIS
LIN {X -2.65,Y -37.7953,Z 60,A -100.9601,B 24.8639,C -2.6924,E1 24.9875,E2 -895.7832} C_DIS
LIN {X -4.5272,Y -37.6166,Z 60,A -104.1626,B 24.8643,C -2.6883,E1 24.9786,E2 -892.569} C_DIS
LIN {X -6.9331,Y -37.2488,Z 60,A -107.6968,B 24.864,C -2.6911,E1 24.9689,E2 -889.0382} C_DIS
LIN {X -9.1032,Y -36.7786,Z 60,A -111.0847,B 24.8639,C -2.6924,E1 24.9597,E2 -885.6489} C_DIS
LIN {X -11.1627,Y -36.2062,Z 60,A -114.3915,B 24.8637,C -2.6937,E1 24.9508,E2 -882.3397} C_DIS
LIN {X -13.4576,Y -35.4178,Z 60,A -118.0902,B 24.8635,C -2.6964,E1 24.9411,E2 -878.6402} C_DIS
LIN {X -16.3875,Y -34.1608,Z 60,A -122.3354,B 24.8623,C -2.7082,E1 24.9303,E2 -874.413} C_DIS
LIN {X -17.7759,Y -33.4598,Z 60,A -125.779,B 24.8632,C -2.6988,E1 24.9217,E2 -870.9373} C_DIS
LIN {X -20.5491,Y -31.8317,Z 60,A -129.6792,B 24.8614,C -2.7165,E1 24.9125,E2 -867.0673} C_DIS
LIN {X -21.9388,Y -30.8904,Z 60,A -132.6519,B 24.8614,C -2.7157,E1 24.9056,E2 -864.0828} C_DIS
LIN {X -23.7813,Y -29.4954,Z 60,A -136.1824,B 24.8609,C -2.7215,E1 24.8978,E2 -860.5529} C_DIS
LIN {X -25.513,Y -28.0111,Z 60,A -139.7288,B 24.8603,C -2.727,E1 24.8904,E2 -857.0057} C_DIS
LIN {X -27.4777,Y -26.0867,Z 60,A -143.6632,B 24.8592,C -2.7379,E1 24.8827,E2 -853.0807} C_DIS
LIN {X -28.8756,Y -24.53,Z 60,A -146.9915,B 24.8587,C -2.7432,E1 24.8766,E2 -849.7501} C_DIS
LIN {X -30.4469,Y -22.5511,Z 60,A -150.7871,B 24.8577,C -2.7524,E1 24.8701,E2 -845.9584} C_DIS
LIN {X -31.6465,Y -20.8333,Z 60,A -154.0791,B 24.857,C -2.759,E1 24.8649,E2 -842.6658} C_DIS
LIN {X -32.8501,Y -18.8784,Z 60,A -157.5283,B 24.8561,C -2.7682,E1 24.86,E2 -839.2207} C_DIS
LIN {X -33.9678,Y -16.7835,Z 60,A -161.0662,B 24.855,C -2.7783,E1 24.8555,E2 -835.6882} C_DIS
LIN {X -35.1667,Y -14.0994,Z 60,A -165.4489,B 24.8536,C -2.7913,E1 24.8507,E2 -831.3124} C_DIS
LIN {X -36.1069,Y -11.4795,Z 60,A -170.4217,B 24.8531,C -2.7962,E1 24.8462,E2 -826.3228} C_DIS
LIN {X -37.0502,Y -7.9239,Z 60,A -175.9333,B 24.8513,C -2.8133,E1 24.8426,E2 -820.82} C_DIS
LIN {X -37.4525,Y -5.73,Z 60,A -179.6028,B 24.8505,C -2.8209,E1 24.841,E2 -817.1467} C_DIS
LIN {X -37.8507,Y -1.6837,Z 60,A 175.3203,B 24.8474,C -2.8499,E1 24.8399,E2 -812.1089} C_DIS
LIN {X -37.8866,Y 0.2479,Z 60,A 172.116,B 24.8467,C -2.8564,E1 24.8399,E2 -808.9008} C_DIS
LIN {X -37.7845,Y 2.7961,Z 60,A 168.2793,B 24.8454,C -2.8687,E1 24.8404,E2 -805.0703} C_DIS
LIN {X -37.5686,Y 4.9102,Z 60,A 164.8671,B 24.8445,C -2.8769,E1 24.8415,E2 -801.6574} C_DIS
LIN {X -37.2348,Y 7.0066,Z 60,A 161.5602,B 24.8435,C -2.886,E1 24.8431,E2 -798.3525} C_DIS
LIN {X -36.6907,Y 9.45,Z 60,A 157.8475,B 24.8422,C -2.8983,E1 24.8455,E2 -794.6477} C_DIS
LIN {X -36.0216,Y 11.746,Z 60,A 153.6581,B 24.8415,C -2.904,E1 24.8489,E2 -790.4478} C_DIS
LIN {X -35.1532,Y 14.133,Z 60,A 150.4532,B 24.8396,C -2.9215,E1 24.8521,E2 -787.2667} C_DIS
LIN {X -34.3348,Y 16.0197,Z 60,A 146.5704,B 24.8394,C -2.9232,E1 24.8567,E2 -783.367} C_DIS
LIN {X -33.0475,Y 18.5308,Z 60,A 142.8551,B 24.8375,C -2.9406,E1 24.8615,E2 -779.6735} C_DIS
LIN {X -31.8015,Y 20.596,Z 60,A 139.1943,B 24.8364,C -2.9506,E1 24.867,E2 -776.0179} C_DIS
LIN {X -30.5069,Y 22.4691,Z 60,A 135.77,B 24.8354,C -2.9599,E1 24.8725,E2 -772.5991} C_DIS
LIN {X -29.0395,Y 24.3358,Z 60,A 132.137,B 24.8344,C -2.9686,E1 24.8789,E2 -768.9702} C_DIS
LIN {X -27.4934,Y 26.0703,Z 60,A 127.9673,B 24.8342,C -2.9706,E1 24.8868,E2 -764.7869} C_DIS
LIN {X -25.5051,Y 28.0178,Z 60,A 124.4855,B 24.8322,C -2.9876,E1 24.8938,E2 -761.3314} C_DIS
LIN {X -24.2775,Y 29.0883,Z 60,A 121.8484,B 24.8318,C -2.9911,E1 24.8995,E2 -758.6926} C_DIS
LIN {X -22.3392,Y 30.602,Z 60,A 118.1555,B 24.831,C -2.999,E1 24.9077,E2 -755.0051} C_DIS
LIN {X -20.4522,Y 31.8941,Z 60,A 114.68,B 24.8302,C -3.0054,E1 24.9157,E2 -751.5334} C_DIS
LIN {X -18.4597,Y 33.0872,Z 60,A 111.1008,B 24.8296,C -3.0107,E1 24.9244,E2 -747.9563} C_DIS
LIN {X -15.4975,Y 34.5736,Z 60,A 106.548,B 24.8282,C -3.0235,E1 24.9358,E2 -743.4222} C_DIS
LIN {X -14.1126,Y 35.1614,Z 60,A 103.6606,B 24.8286,C -3.0198,E1 24.9433,E2 -740.5195} C_DIS
LIN {X -11.6261,Y 36.0601,Z 60,A 99.81,B 24.8279,C -3.0262,E1 24.9534,E2 -736.677} C_DIS
LIN {X -9.2605,Y 36.7386,Z 60,A 96.4196,B 24.827,C -3.0338,E1 24.9625,E2 -733.2994} C_DIS
LIN {X -7.6937,Y 37.0989,Z 60,A 93.7992,B 24.827,C -3.0337,E1 24.9697,E2 -730.6754} C_DIS
LIN {X -5.7249,Y 37.4533,Z 60,A 90.6284,B 24.827,C -3.0341,E1 24.9784,E2 -727.5025} C_DIS
LIN {X -3.3516,Y 37.74,Z 60,A 86.9185,B 24.8269,C -3.0348,E1 24.9887,E2 -723.7922} C_DIS
LIN {X -0.606,Y 37.8836,Z 60,A 83.2497,B 24.826,C -3.0421,E1 24.9989,E2 -720.14} C_DIS
LIN {X 1.0217,Y 37.8745,Z 60,A 80.4607,B 24.8265,C -3.0384,E1 25.0067,E2 -717.3427} C_DIS
LIN {X 3.3569,Y 37.7395,Z 60,A 76.8536,B 24.8265,C -3.0374,E1 25.0168,E2 -713.7348} C_DIS
LIN {X 5.6358,Y 37.4671,Z 60,A 73.344,B 24.8267,C -3.0362,E1 25.0265,E2 -710.2251} C_DIS
LIN {X 7.9872,Y 37.0365,Z 60,A 69.8032,B 24.8267,C -3.0356,E1 25.0362,E2 -706.6873} C_DIS
LIN {X 10.2936,Y 36.4629,Z 60,A 66.0859,B 24.8272,C -3.0318,E1 25.0462,E2 -702.9668} C_DIS
LIN {X 13.3407,Y 35.4615,Z 60,A 61.3169,B 24.8276,C -3.0288,E1 25.0588,E2 -698.2002} C_DIS
LIN {X 15.5774,Y 34.5377,Z 60,A 57.3934,B 24.8284,C -3.0214,E1 25.0689,E2 -694.2684} C_DIS
LIN {X 17.9313,Y 33.3767,Z 60,A 53.7686,B 24.8284,C -3.0211,E1 25.0778,E2 -690.653} C_DIS
LIN {X 19.85,Y 32.2725,Z 60,A 50.3467,B 24.8291,C -3.0153,E1 25.086,E2 -687.2278} C_DIS
LIN {X 21.8193,Y 30.9749,Z 60,A 46.7807,B 24.8298,C -3.0096,E1 25.0943,E2 -683.6605} C_DIS
LIN {X 23.7232,Y 29.5425,Z 60,A 43.2626,B 24.8303,C -3.0044,E1 25.102,E2 -680.1431} C_DIS
LIN {X 25.5584,Y 27.9694,Z 60,A 39.592,B 24.8312,C -2.9972,E1 25.1097,E2 -676.4699} C_DIS
LIN {X 27.1234,Y 26.4552,Z 60,A 36.2548,B 24.832,C -2.9898,E1 25.1163,E2 -673.1291} C_DIS
LIN {X 28.7317,Y 24.6984,Z 60,A 32.8528,B 24.8326,C -2.9848,E1 25.1226,E2 -669.7305} C_DIS
LIN {X 30.5498,Y 22.4106,Z 60,A 28.48,B 24.8337,C -2.9751,E1 25.1301,E2 -665.3555} C_DIS
LIN {X 31.784,Y 20.6231,Z 60,A 25.0638,B 24.8348,C -2.9649,E1 25.1354,E2 -661.9322} C_DIS
LIN {X 32.959,Y 18.6888,Z 60,A 21.5118,B 24.836,C -2.9541,E1 25.1404,E2 -658.3726} C_DIS
LIN {X 33.8421,Y 17.0376,Z 60,A 18.8591,B 24.8365,C -2.9492,E1 25.1438,E2 -655.7225} C_DIS
LIN {X 34.7718,Y 15.0469,Z 60,A 15.5806,B 24.8375,C -2.9407,E1 25.1476,E2 -652.4417} C_DIS
LIN {X 35.5679,Y 13.0556,Z 60,A 12.3198,B 24.8385,C -2.9312,E1 25.1508,E2 -649.1765} C_DIS
LIN {X 36.5088,Y 10.1288,Z 60,A 7.5202,B 24.8403,C -2.9152,E1 25.1547,E2 -644.3664} C_DIS
LIN {X 37.0988,Y 7.6945,Z 60,A 4.0355,B 24.841,C -2.9085,E1 25.1569,E2 -640.8862} C_DIS
LIN {X 37.4621,Y 5.6681,Z 60,A 0.9106,B 24.8421,C -2.8988,E1 25.1583,E2 -637.7567} C_DIS
LIN {X 37.7343,Y 3.4125,Z 60,A -2.8413,B 24.8438,C -2.8833,E1 25.1594,E2 -633.9901} C_DIS
LIN {X 37.8552,Y 1.5766,Z 60,A -5.3474,B 24.8443,C -2.8789,E1 25.1597,E2 -631.4887} C_DIS
LIN {X 37.8753,Y -0.9935,Z 60,A -9.8029,B 24.8466,C -2.8578,E1 25.1596,E2 -627.0097} C_DIS
LIN {X 37.7361,Y -3.3939,Z 60,A -13.5863,B 24.848,C -2.8441,E1 25.1587,E2 -623.2163} C_DIS
LIN {X 37.362,Y -6.2931,Z 60,A -17.1782,B 24.8481,C -2.8433,E1 25.1572,E2 -619.6436} C_DIS
LIN {X 36.9049,Y -8.5758,Z 60,A -20.6087,B 24.8491,C -2.8338,E1 25.1551,E2 -616.2105} C_DIS
LIN {X 36.1919,Y -11.2094,Z 60,A -24.7629,B 24.8505,C -2.8207,E1 25.1519,E2 -612.0491} C_DIS
LIN {X 35.4314,Y -13.4211,Z 60,A -28.281,B 24.8516,C -2.8103,E1 25.1486,E2 -608.5261} C_DIS
LIN {X 34.5247,Y -15.6064,Z 60,A -31.809,B 24.8527,C -2.8005,E1 25.1447,E2 -604.9941} C_DIS
LIN {X 33.5824,Y -17.5422,Z 60,A -35.0697,B 24.8537,C -2.791,E1 25.1406,E2 -601.7283} C_DIS
LIN {X 31.9981,Y -20.289,Z 60,A -39.8538,B 24.8551,C -2.7777,E1 25.1337,E2 -596.9373} C_DIS
LIN {X 30.664,Y -22.2541,Z 60,A -43.4626,B 24.8561,C -2.7678,E1 25.1279,E2 -593.3227} C_DIS
LIN {X 29.1818,Y -24.165,Z 60,A -47.048,B 24.857,C -2.7594,E1 25.1217,E2 -589.7342} C_DIS
LIN {X 27.6371,Y -25.9175,Z 60,A -50.5768,B 24.8579,C -2.7508,E1 25.115,E2 -586.2005} C_DIS
LIN {X 25.856,Y -27.6947,Z 60,A -54.1441,B 24.8584,C -2.7454,E1 25.1079,E2 -582.6354} C_DIS
LIN {X 24.7267,Y -28.7074,Z 60,A -56.554,B 24.8591,C -2.7386,E1 25.1028,E2 -580.2189} C_DIS
LIN {X 22.9507,Y -30.1465,Z 60,A -60.1253,B 24.8601,C -2.7296,E1 25.095,E2 -576.6394} C_DIS
LIN {X 20.9903,Y -31.5426,Z 60,A -63.7444,B 24.8608,C -2.7227,E1 25.0866,E2 -573.0165} C_DIS
LIN {X 18.9093,Y -32.8323,Z 60,A -67.3783,B 24.8614,C -2.717,E1 25.0779,E2 -569.3804} C_DIS
LIN {X 16.7766,Y -33.9712,Z 60,A -71.4489,B 24.8626,C -2.7052,E1 25.0677,E2 -565.2929} C_DIS
LIN {X 14.4352,Y -35.031,Z 60,A -74.8879,B 24.8625,C -2.7059,E1 25.0589,E2 -561.8636} C_DIS
LIN {X 12.3822,Y -35.8076,Z 60,A -78.1586,B 24.8629,C -2.7023,E1 25.0504,E2 -558.5913} C_DIS
LIN {X 10.1371,Y -36.5066,Z 60,A -81.754,B 24.8633,C -2.6978,E1 25.0407,E2 -554.9915} C_DIS
LIN {X 7.8526,Y -37.0656,Z 60,A -85.8949,B 24.8644,C -2.6867,E1 25.0294,E2 -550.8297} C_DIS
LIN {X 4.6326,Y -37.604,Z 60,A -90.2534,B 24.864,C -2.6911,E1 25.0174,E2 -546.4855} C_DIS
LIN {X 2.2685,Y -37.8199,Z 60,A -93.8226,B 24.8641,C -2.6897,E1 25.0074,E2 -542.9148} C_DIS
LIN {X 0.1475,Y -37.8851,Z 60,A -95.6528,B 24.8624,C -2.7068,E1 25.0025,E2 -541.1256} C_DIS
Enddeposition()
LIN {X 0.1475,Y -37.8851,Z 60,A -95.6528,B 24.8624,C -2.7068,E1 25.0025,E2 -541.1256} C_DIS
Startdeposition()
$VEL.CP = VEL_PRINT
LIN {X 0.7723,Y -36.9222,Z 60,A -94.3417,B 24.8602,C -2.7279,E1 25.0062,E2 -542.4866} C_DIS
LIN {X 3.0934,Y -36.8,Z 60,A -90.7795,B 24.8602,C -2.7289,E1 25.0162,E2 -546.0497} C_DIS
LIN {X 4.7976,Y -36.617,Z 60,A -88.1793,B 24.8601,C -2.7297,E1 25.0234,E2 -548.6497} C_DIS
LIN {X 6.6439,Y -36.3272,Z 60,A -85.2458,B 24.8598,C -2.7324,E1 25.0315,E2 -551.5865} C_DIS
LIN {X 8.8043,Y -35.8653,Z 60,A -81.8058,B 24.8594,C -2.7357,E1 25.0408,E2 -555.0297} C_DIS
LIN {X 11.3429,Y -35.1448,Z 60,A -77.7138,B 24.859,C -2.7403,E1 25.0518,E2 -559.1253} C_DIS
LIN {X 13.2715,Y -34.4631,Z 60,A -73.9077,B 24.8576,C -2.7534,E1 25.0618,E2 -562.9543} C_DIS
LIN {X 16.5872,Y -32.9961,Z 60,A -69.2356,B 24.8581,C -2.7483,E1 25.0735,E2 -567.6026} C_DIS
LIN {X 18.2686,Y -32.0955,Z 60,A -66.0204,B 24.8572,C -2.7571,E1 25.0814,E2 -570.8291} C_DIS
LIN {X 20.1563,Y -30.9448,Z 60,A -62.5156,B 24.8564,C -2.7646,E1 25.0897,E2 -574.3403} C_DIS
LIN {X 22.096,Y -29.5907,Z 60,A -58.903,B 24.8558,C -2.7711,E1 25.0979,E2 -577.9558} C_DIS
LIN {X 23.8427,Y -28.2025,Z 60,A -55.4488,B 24.855,C -2.7785,E1 25.1053,E2 -581.4143} C_DIS
LIN {X 25.3058,Y -26.8971,Z 60,A -52.7298,B 24.8548,C -2.7806,E1 25.1109,E2 -584.1273} C_DIS
LIN {X 26.7862,Y -25.4237,Z 60,A -49.2219,B 24.8535,C -2.7924,E1 25.1178,E2 -587.6482} C_DIS
LIN {X 28.3179,Y -23.7052,Z 60,A -45.6391,B 24.8526,C -2.8015,E1 25.1243,E2 -591.2364} C_DIS
LIN {X 29.7811,Y -21.8385,Z 60,A -42.0951,B 24.8518,C -2.8091,E1 25.1303,E2 -594.7816} C_DIS
LIN {X 31.0151,Y -20.0472,Z 60,A -38.8593,B 24.851,C -2.8162,E1 25.1354,E2 -598.018} C_DIS
LIN {X 32.0794,Y -18.2966,Z 60,A -35.5009,B 24.8498,C -2.8279,E1 25.1401,E2 -601.3868} C_DIS
LIN {X 33.0247,Y -16.528,Z 60,A -32.267,B 24.8486,C -2.8388,E1 25.1443,E2 -604.6294} C_DIS
LIN {X 34.0897,Y -14.2027,Z 60,A -28.441,B 24.8476,C -2.8483,E1 25.1485,E2 -608.457} C_DIS
LIN {X 34.7133,Y -12.6017,Z 60,A -25.3731,B 24.846,C -2.8627,E1 25.1515,E2 -611.5417} C_DIS
LIN {X 35.6898,Y -9.4893,Z 60,A -21.2478,B 24.846,C -2.8634,E1 25.1548,E2 -615.6453} C_DIS
LIN {X 36.0802,Y -7.8766,Z 60,A -18.2126,B 24.8443,C -2.8787,E1 25.1567,E2 -618.6989} C_DIS
LIN {X 36.5186,Y -5.5003,Z 60,A -14.0125,B 24.8422,C -2.8975,E1 25.1585,E2 -622.9189} C_DIS
LIN {X 36.8189,Y -2.8621,Z 60,A -10.295,B 24.8415,C -2.9041,E1 25.1595,E2 -626.6299} C_DIS
LIN {X 36.9253,Y -0.6026,Z 60,A -6.4409,B 24.8397,C -2.9205,E1 25.1598,E2 -630.5001} C_DIS
LIN {X 36.8926,Y 1.6648,Z 60,A -3.3171,B 24.8392,C -2.9252,E1 25.1595,E2 -633.6165} C_DIS
LIN {X 36.6424,Y 4.6037,Z 60,A 1.1223,B 24.8379,C -2.9372,E1 25.1582,E2 -638.0579} C_DIS
LIN {X 36.2815,Y 6.8906,Z 60,A 4.6456,B 24.8368,C -2.9471,E1 25.1565,E2 -641.584} C_DIS
LIN {X 35.6927,Y 9.478,Z 60,A 8.6557,B 24.8356,C -2.9577,E1 25.1539,E2 -645.596} C_DIS
LIN {X 35.1736,Y 11.2527,Z 60,A 11.3154,B 24.835,C -2.9629,E1 25.1517,E2 -648.2528} C_DIS
LIN {X 34.5493,Y 13.0442,Z 60,A 14.854,B 24.833,C -2.9806,E1 25.1483,E2 -651.8135} C_DIS
LIN {X 33.3577,Y 15.8464,Z 60,A 19.4975,B 24.8317,C -2.9924,E1 25.1429,E2 -656.4597} C_DIS
LIN {X 32.0978,Y 18.2645,Z 60,A 23.6802,B 24.8305,C -3.0028,E1 25.1373,E2 -660.6453} C_DIS
LIN {X 30.6996,Y 20.5275,Z 60,A 27.5678,B 24.8298,C -3.0096,E1 25.1314,E2 -664.5294} C_DIS
LIN {X 29.0079,Y 22.8557,Z 60,A 31.8211,B 24.8289,C -3.017,E1 25.1243,E2 -668.78} C_DIS
LIN {X 27.646,Y 24.4857,Z 60,A 34.8501,B 24.8285,C -3.0205,E1 25.1188,E2 -671.8035} C_DIS
LIN {X 26.0339,Y 26.193,Z 60,A 38.859,B 24.827,C -3.0335,E1 25.111,E2 -675.8261} C_DIS
LIN {X 24.5446,Y 27.5934,Z 60,A 42.7472,B 24.8251,C -3.0501,E1 25.1029,E2 -679.738} C_DIS
LIN {X 21.9898,Y 29.6703,Z 60,A 47.1379,B 24.8253,C -3.0488,E1 25.0933,E2 -684.1094} C_DIS
LIN {X 20.133,Y 30.9599,Z 60,A 50.675,B 24.8246,C -3.0547,E1 25.0851,E2 -687.6488} C_DIS
LIN {X 18.5321,Y 31.944,Z 60,A 53.5153,B 24.8242,C -3.0578,E1 25.0782,E2 -690.4877} C_DIS
LIN {X 16.926,Y 32.823,Z 60,A 56.6363,B 24.8234,C -3.0653,E1 25.0705,E2 -693.6178} C_DIS
LIN {X 14.0497,Y 34.1526,Z 60,A 61.0683,B 24.8235,C -3.0641,E1 25.0592,E2 -698.036} C_DIS
LIN {X 12.3285,Y 34.8114,Z 60,A 63.8744,B 24.8233,C -3.0659,E1 25.0519,E2 -700.8405} C_DIS
LIN {X 10.7528,Y 35.3299,Z 60,A 66.5521,B 24.8229,C -3.0692,E1 25.0447,E2 -703.5212} C_DIS
LIN {X 9.0215,Y 35.8109,Z 60,A 69.9565,B 24.8218,C -3.079,E1 25.0355,E2 -706.9436} C_DIS
LIN {X 6.1192,Y 36.4197,Z 60,A 74.0386,B 24.8223,C -3.0741,E1 25.0243,E2 -711.0093} C_DIS
LIN {X 4.0775,Y 36.7047,Z 60,A 77.3495,B 24.8221,C -3.0761,E1 25.0151,E2 -714.3225} C_DIS
LIN {X 1.9625,Y 36.8778,Z 60,A 80.9295,B 24.8217,C -3.0797,E1 25.0051,E2 -717.9096} C_DIS
LIN {X -0.782,Y 36.922,Z 60,A 84.9177,B 24.8222,C -3.0755,E1 24.994,E2 -721.8876} C_DIS
LIN {X -3.5894,Y 36.7552,Z 60,A 89.1325,B 24.8226,C -3.0718,E1 24.9823,E2 -726.0955} C_DIS
LIN {X -5.884,Y 36.459,Z 60,A 92.8359,B 24.8227,C -3.0708,E1 24.9721,E2 -729.7997} C_DIS
LIN {X -7.4749,Y 36.1657,Z 60,A 95.7302,B 24.8224,C -3.0733,E1 24.9641,E2 -732.7032} C_DIS
LIN {X -10.7173,Y 35.3406,Z 60,A 100.1551,B 24.8241,C -3.0593,E1 24.9523,E2 -737.1014} C_DIS
LIN {X -12.1378,Y 34.878,Z 60,A 102.7991,B 24.824,C -3.0602,E1 24.9453,E2 -739.7527} C_DIS
LIN {X -14.2493,Y 34.0701,Z 60,A 106.3439,B 24.8245,C -3.0559,E1 24.9361,E2 -743.295} C_DIS
LIN {X -17.1077,Y 32.7284,Z 60,A 112.0529,B 24.8243,C -3.0571,E1 24.9218,E2 -749.022} C_DIS
LIN {X -20.1077,Y 30.9762,Z 60,A 116.7267,B 24.8263,C -3.0397,E1 24.9107,E2 -753.6687} C_DIS
LIN {X -22.0361,Y 29.6356,Z 60,A 120.4102,B 24.8271,C -3.0329,E1 24.9024,E2 -757.3488} C_DIS
LIN {X -23.4762,Y 28.5084,Z 60,A 123.8468,B 24.8271,C -3.033,E1 24.895,E2 -760.7988} C_DIS
LIN {X -26.1813,Y 26.0459,Z 60,A 128.5582,B 24.8297,C -3.0102,E1 24.8855,E2 -765.475} C_DIS
LIN {X -27.1462,Y 25.0386,Z 60,A 131.3198,B 24.8296,C -3.011,E1 24.8802,E2 -768.2505} C_DIS
LIN {X -29.2617,Y 22.5298,Z 60,A 136.1999,B 24.8313,C -2.9959,E1 24.8716,E2 -773.1172} C_DIS
LIN {X -30.6534,Y 20.5966,Z 60,A 140.1476,B 24.8321,C -2.9884,E1 24.8653,E2 -777.0666} C_DIS
LIN {X -32.046,Y 18.3546,Z 60,A 143.8492,B 24.8339,C -2.9732,E1 24.8601,E2 -780.7509} C_DIS
LIN {X -33.1427,Y 16.2904,Z 60,A 147.9312,B 24.8345,C -2.9672,E1 24.8549,E2 -784.8403} C_DIS
LIN {X -34.1872,Y 13.9668,Z 60,A 151.4757,B 24.8363,C -2.9517,E1 24.851,E2 -788.3672} C_DIS
LIN {X -34.7047,Y 12.6249,Z 60,A 154.0375,B 24.8367,C -2.9481,E1 24.8485,E2 -790.935} C_DIS
LIN {X -35.5343,Y 10.0566,Z 60,A 158.2236,B 24.8381,C -2.9353,E1 24.8451,E2 -795.1146} C_DIS
LIN {X -36.131,Y 7.6414,Z 60,A 162.0023,B 24.8395,C -2.9226,E1 24.8428,E2 -798.885} C_DIS
LIN {X -36.5317,Y 5.4136,Z 60,A 165.1438,B 24.8411,C -2.9082,E1 24.8413,E2 -802.0107} C_DIS
LIN {X -36.7374,Y 3.761,Z 60,A 167.8837,B 24.8418,C -2.9016,E1 24.8404,E2 -804.7512} C_DIS
LIN {X -36.8802,Y 1.9049,Z 60,A 171.3672,B 24.8422,C -2.8981,E1 24.8399,E2 -808.2473} C_DIS
LIN {X -36.9284,Y 0.0318,Z 60,A 174.6718,B 24.8428,C -2.8928,E1 24.8399,E2 -811.5592} C_DIS
LIN {X -36.828,Y -2.7396,Z 60,A 178.2369,B 24.845,C -2.8725,E1 24.8404,E2 -815.0969} C_DIS
LIN {X -36.6116,Y -4.8387,Z 60,A -178.4963,B 24.8461,C -2.8623,E1 24.8415,E2 -818.3589} C_DIS
LIN {X -36.2847,Y -6.8732,Z 60,A -175.2585,B 24.8471,C -2.853,E1 24.843,E2 -821.5937} C_DIS
LIN {X -35.8662,Y -8.8001,Z 60,A -172.452,B 24.8483,C -2.8414,E1 24.8448,E2 -824.389} C_DIS
LIN {X -35.554,Y -9.9861,Z 60,A -170.1114,B 24.8485,C -2.84,E1 24.8465,E2 -826.7396} C_DIS
LIN {X -34.7183,Y -12.5877,Z 60,A -165.6906,B 24.8496,C -2.8295,E1 24.8505,E2 -831.1606} C_DIS
LIN {X -33.7191,Y -15.0613,Z 60,A -161.4276,B 24.8507,C -2.8191,E1 24.8552,E2 -835.4224} C_DIS
LIN {X -32.4707,Y -17.5924,Z 60,A -157.3723,B 24.8523,C -2.8042,E1 24.8604,E2 -839.4637} C_DIS
LIN {X -31.3418,Y -19.5329,Z 60,A -153.8212,B 24.8532,C -2.7959,E1 24.8655,E2 -843.0132} C_DIS
LIN {X -29.8421,Y -21.755,Z 60,A -149.4795,B 24.854,C -2.7876,E1 24.8724,E2 -847.3565} C_DIS
LIN {X -28.1978,Y -23.8482,Z 60,A -145.4005,B 24.8551,C -2.7777,E1 24.8796,E2 -851.4307} C_DIS
LIN {X -26.4339,Y -25.7896,Z 60,A -141.3961,B 24.8561,C -2.7683,E1 24.8872,E2 -855.4302} C_DIS
LIN {X -24.524,Y -27.6121,Z 60,A -137.2112,B 24.8568,C -2.7612,E1 24.8958,E2 -859.6152} C_DIS
LIN {X -22.7053,Y -29.1265,Z 60,A -133.5182,B 24.8575,C -2.7549,E1 24.9039,E2 -863.3069} C_DIS
LIN {X -21.3239,Y -30.1519,Z 60,A -130.7818,B 24.8578,C -2.7513,E1 24.9101,E2 -866.0441} C_DIS
LIN {X -19.4098,Y -31.4182,Z 60,A -127.4765,B 24.8587,C -2.7431,E1 24.9178,E2 -869.3405} C_DIS
LIN {X -17.6935,Y -32.4154,Z 60,A -124.5856,B 24.8593,C -2.7369,E1 24.9248,E2 -872.225} C_DIS
LIN {X -15.9632,Y -33.3017,Z 60,A -121.2863,B 24.8593,C -2.7365,E1 24.9331,E2 -875.5321} C_DIS
LIN {X -14.1248,Y -34.1213,Z 60,A -118.5504,B 24.8601,C -2.7288,E1 24.9401,E2 -878.2562} C_DIS
LIN {X -12.9362,Y -34.5898,Z 60,A -116.219,B 24.8599,C -2.7311,E1 24.9462,E2 -880.5978} C_DIS
LIN {X -10.863,Y -35.296,Z 60,A -112.7097,B 24.86,C -2.7298,E1 24.9555,E2 -884.1106} C_DIS
LIN {X -8.6505,Y -35.9023,Z 60,A -109.231,B 24.8603,C -2.7269,E1 24.9649,E2 -887.5873} C_DIS
LIN {X -6.4823,Y -36.3569,Z 60,A -105.1316,B 24.8596,C -2.7338,E1 24.9762,E2 -891.7076} C_DIS
LIN {X -3.3088,Y -36.7817,Z 60,A -100.9258,B 24.8607,C -2.7236,E1 24.9878,E2 -895.8918} C_DIS
LIN {X -0.4133,Y -36.9283,Z 60,A -96.1691,B 24.8603,C -2.7274,E1 25.0011,E2 -900.6584} C_DIS
LIN {X -0.4133,Y -36.9283,Z 60,A -96.1691,B 24.8603,C -2.7274,E1 25.0011,E2 -900.6584} C_DIS
Enddeposition()
LIN {X 0.1425,Y -35.9633,Z 60,A -96.4696,B 24.8601,C -2.7295,E1 25.0003,E2 -900.363} C_DIS
Startdeposition()
$VEL.CP = VEL_PRINT
LIN {X -2.4905,Y -35.8856,Z 60,A -101.4433,B 24.8611,C -2.7196,E1 24.9864,E2 -895.3645} C_DIS
LIN {X -4.708,Y -35.6625,Z 60,A -104.9383,B 24.861,C -2.7207,E1 24.9767,E2 -891.8699} C_DIS
LIN {X -7.2145,Y -35.2409,Z 60,A -108.568,B 24.8603,C -2.7269,E1 24.9667,E2 -888.2513} C_DIS
LIN {X -9.1945,Y -34.7767,Z 60,A -112.2847,B 24.8607,C -2.7232,E1 24.9566,E2 -884.5205} C_DIS
LIN {X -11.7275,Y -34.0065,Z 60,A -115.9407,B 24.8598,C -2.7326,E1 24.9469,E2 -880.8804} C_DIS
LIN {X -13.7816,Y -33.2273,Z 60,A -120.2602,B 24.8603,C -2.7269,E1 24.9357,E2 -876.5378} C_DIS
LIN {X -16.1353,Y -32.1506,Z 60,A -124.2063,B 24.8597,C -2.7335,E1 24.9258,E2 -872.5974} C_DIS
LIN {X -18.4556,Y -30.8773,Z 60,A -127.9898,B 24.8586,C -2.7438,E1 24.9166,E2 -868.8273} C_DIS
LIN {X -19.7397,Y -30.0721,Z 60,A -131.1605,B 24.859,C -2.7396,E1 24.9091,E2 -865.6363} C_DIS
LIN {X -22.1387,Y -28.3533,Z 60,A -135.733,B 24.8581,C -2.7489,E1 24.8989,E2 -861.0696} C_DIS
LIN {X -24.068,Y -26.7344,Z 60,A -139.2456,B 24.8568,C -2.7614,E1 24.8916,E2 -857.5731} C_DIS
LIN {X -25.3816,Y -25.4901,Z 60,A -141.988,B 24.856,C -2.7686,E1 24.8861,E2 -854.8366} C_DIS
LIN {X -26.5782,Y -24.2404,Z 60,A -145.1521,B 24.8558,C -2.7705,E1 24.88,E2 -851.6631} C_DIS
LIN {X -28.1018,Y -22.4558,Z 60,A -148.4091,B 24.8545,C -2.7836,E1 24.8742,E2 -848.4223} C_DIS
LIN {X -29.5373,Y -20.5313,Z 60,A -153.3773,B 24.8546,C -2.782,E1 24.8661,E2 -843.4262} C_DIS
LIN {X -30.7792,Y -18.6182,Z 60,A -156.6611,B 24.8533,C -2.7945,E1 24.8613,E2 -840.1554} C_DIS
LIN {X -32.0955,Y -16.2444,Z 60,A -160.5227,B 24.8516,C -2.8102,E1 24.8563,E2 -836.3109} C_DIS
LIN {X -33.2615,Y -13.6998,Z 60,A -165.7895,B 24.8511,C -2.8153,E1 24.8504,E2 -831.0273} C_DIS
LIN {X -34.2894,Y -10.8714,Z 60,A -169.686,B 24.8488,C -2.8372,E1 24.8469,E2 -827.1608} C_DIS
LIN {X -34.7584,Y -9.2633,Z 60,A -172.6948,B 24.8483,C -2.842,E1 24.8446,E2 -824.1462} C_DIS
LIN {X -35.4595,Y -6.0522,Z 60,A -177.6436,B 24.8463,C -2.8603,E1 24.8418,E2 -819.2121} C_DIS
LIN {X -35.7501,Y -3.9888,Z 60,A 178.9783,B 24.8452,C -2.87,E1 24.8406,E2 -815.8369} C_DIS
LIN {X -35.8803,Y -2.5624,Z 60,A 176.4343,B 24.8447,C -2.8748,E1 24.84,E2 -813.2891} C_DIS
LIN {X -35.97,Y -0.371,Z 60,A 172.9193,B 24.8436,C -2.8855,E1 24.8398,E2 -809.7785} C_DIS
LIN {X -35.93,Y 1.7308,Z 60,A 169.4982,B 24.8425,C -2.8953,E1 24.8401,E2 -806.3604} C_DIS
LIN {X -35.7,Y 4.4162,Z 60,A 164.8226,B 24.8414,C -2.9055,E1 24.8415,E2 -801.681} C_DIS
LIN {X -35.0433,Y 8.1192,Z 60,A 158.5869,B 24.8396,C -2.922,E1 24.8449,E2 -795.448} C_DIS
LIN {X -34.3105,Y 10.8051,Z 60,A 154.7261,B 24.8375,C -2.9405,E1 24.8479,E2 -791.6092} C_DIS
LIN {X -33.6546,Y 12.7016,Z 60,A 151.4023,B 24.8366,C -2.949,E1 24.8511,E2 -788.2869} C_DIS
LIN {X -32.8787,Y 14.5941,Z 60,A 147.5858,B 24.8361,C -2.9537,E1 24.8553,E2 -784.4606} C_DIS
LIN {X -31.6023,Y 17.1838,Z 60,A 143.6745,B 24.8339,C -2.9729,E1 24.8603,E2 -780.5745} C_DIS
LIN {X -30.5355,Y 19.0148,Z 60,A 139.8445,B 24.8333,C -2.9782,E1 24.8658,E2 -776.7374} C_DIS
LIN {X -28.9896,Y 21.2977,Z 60,A 134.943,B 24.8325,C -2.9853,E1 24.8738,E2 -771.829} C_DIS
LIN {X -26.0956,Y 24.7594,Z 60,A 127.4239,B 24.8308,C -3,E1 24.8878,E2 -764.3114} C_DIS
LIN {X -22.6383,Y 27.9552,Z 60,A 121.3313,B 24.8274,C -3.03,E1 24.9004,E2 -758.2663} C_DIS
LIN {X -20.5704,Y 29.5101,Z 60,A 116.1535,B 24.8277,C -3.0279,E1 24.9121,E2 -753.0655} C_DIS
LIN {X -18.2458,Y 31.0014,Z 60,A 111.8227,B 24.8267,C -3.0364,E1 24.9225,E2 -748.7416} C_DIS
LIN {X -15.1472,Y 32.6271,Z 60,A 106.9867,B 24.8248,C -3.0527,E1 24.9345,E2 -743.9316} C_DIS
LIN {X -13.4829,Y 33.3492,Z 60,A 104.3221,B 24.8241,C -3.0591,E1 24.9413,E2 -741.2762} C_DIS
LIN {X -12.2872,Y 33.8081,Z 60,A 102.0017,B 24.8241,C -3.0587,E1 24.9474,E2 -738.9501} C_DIS
LIN {X -10.5136,Y 34.4009,Z 60,A 99.2732,B 24.8234,C -3.0648,E1 24.9546,E2 -736.2311} C_DIS
LIN {X -8.7008,Y 34.9037,Z 60,A 95.5652,B 24.824,C -3.06,E1 24.9647,E2 -732.5063} C_DIS
LIN {X -6.2267,Y 35.4293,Z 60,A 91.7827,B 24.8233,C -3.0659,E1 24.975,E2 -728.7336} C_DIS
LIN {X -3.8481,Y 35.7655,Z 60,A 88.3613,B 24.8225,C -3.0727,E1 24.9844,E2 -725.3259} C_DIS
LIN {X -2.6058,Y 35.877,Z 60,A 85.59,B 24.8234,C -3.0646,E1 24.9922,E2 -722.5343} C_DIS
LIN {X -0.5373,Y 35.9682,Z 60,A 82.4068,B 24.8232,C -3.0668,E1 25.0011,E2 -719.3559} C_DIS
LIN {X 1.8591,Y 35.9236,Z 60,A 79.0831,B 24.8225,C -3.0729,E1 25.0103,E2 -716.0476} C_DIS
LIN {X 3.6093,Y 35.7906,Z 60,A 76.2692,B 24.8225,C -3.0724,E1 25.0182,E2 -713.2342} C_DIS
LIN {X 5.161,Y 35.5999,Z 60,A 73.0555,B 24.8236,C -3.0632,E1 25.0271,E2 -710.0013} C_DIS
LIN {X 8.6391,Y 34.9192,Z 60,A 68.2945,B 24.8227,C -3.0714,E1 25.04,E2 -705.2659} C_DIS
LIN {X 10.8626,Y 34.2923,Z 60,A 63.8769,B 24.824,C -3.0596,E1 25.0519,E2 -700.8279} C_DIS
LIN {X 13.1996,Y 33.4626,Z 60,A 60.216,B 24.824,C -3.0596,E1 25.0614,E2 -697.1749} C_DIS
LIN {X 15.728,Y 32.3516,Z 60,A 55.6102,B 24.8249,C -3.0519,E1 25.0731,E2 -692.5626} C_DIS
LIN {X 18.3343,Y 30.949,Z 60,A 51.6292,B 24.8245,C -3.0552,E1 25.0828,E2 -688.6011} C_DIS
LIN {X 19.8983,Y 29.9676,Z 60,A 48.2675,B 24.8257,C -3.0451,E1 25.0907,E2 -685.2263} C_DIS
LIN {X 21.9005,Y 28.537,Z 60,A 44.6931,B 24.8259,C -3.0432,E1 25.0987,E2 -681.6601} C_DIS
LIN {X 23.5234,Y 27.2147,Z 60,A 40.886,B 24.8274,C -3.0305,E1 25.1069,E2 -677.8375} C_DIS
LIN {X 25.6507,Y 25.2197,Z 60,A 36.5528,B 24.828,C -3.0254,E1 25.1156,E2 -673.5103} C_DIS
LIN {X 27.0792,Y 23.6793,Z 60,A 33.5359,B 24.8283,C -3.0227,E1 25.1212,E2 -670.5005} C_DIS
LIN {X 27.8937,Y 22.7141,Z 60,A 31.0724,B 24.8295,C -3.0117,E1 25.1256,E2 -668.0222} C_DIS
LIN {X 29.3768,Y 20.7604,Z 60,A 27.1894,B 24.8305,C -3.0027,E1 25.1321,E2 -664.1366} C_DIS
LIN {X 30.7926,Y 18.5954,Z 60,A 23.3451,B 24.8313,C -2.9963,E1 25.1378,E2 -660.2964} C_DIS
LIN {X 31.6484,Y 17.0988,Z 60,A 20.573,B 24.8321,C -2.9886,E1 25.1416,E2 -657.5206} C_DIS
LIN {X 32.628,Y 15.1451,Z 60,A 17.5395,B 24.8325,C -2.9858,E1 25.1453,E2 -654.4966} C_DIS
LIN {X 33.2434,Y 13.7423,Z 60,A 14.5778,B 24.8341,C -2.9712,E1 25.1486,E2 -651.5167} C_DIS
LIN {X 33.8726,Y 12.109,Z 60,A 11.9118,B 24.8348,C -2.9651,E1 25.1511,E2 -648.851} C_DIS
LIN {X 34.3019,Y 10.8325,Z 60,A 9.1961,B 24.8364,C -2.9503,E1 25.1535,E2 -646.1158} C_DIS
LIN {X 35.2007,Y 7.4099,Z 60,A 4.5627,B 24.8366,C -2.9485,E1 25.1565,E2 -641.5048} C_DIS
LIN {X 35.5055,Y 5.7767,Z 60,A 1.0002,B 24.839,C -2.9267,E1 25.1582,E2 -637.9116} C_DIS
LIN {X 35.8046,Y 3.462,Z 60,A -3.11,B 24.841,C -2.9093,E1 25.1594,E2 -633.7847} C_DIS
LIN {X 35.9704,Y -0.2276,Z 60,A -8.2886,B 24.8418,C -2.9015,E1 25.1597,E2 -628.6185} C_DIS
LIN {X 35.8842,Y -2.5098,Z 60,A -12.0213,B 24.8432,C -2.8887,E1 25.1591,E2 -624.8775} C_DIS
LIN {X 35.5705,Y -5.3613,Z 60,A -15.9632,B 24.8437,C -2.8839,E1 25.1578,E2 -620.9474} C_DIS
LIN {X 35.2495,Y -7.1723,Z 60,A -19.4146,B 24.8456,C -2.8669,E1 25.1559,E2 -617.476} C_DIS
LIN {X 34.7294,Y -9.3722,Z 60,A -23.1148,B 24.8469,C -2.8543,E1 25.1534,E2 -613.7673} C_DIS
LIN {X 33.7205,Y -12.5255,Z 60,A -27.8485,B 24.8478,C -2.8464,E1 25.1491,E2 -609.0416} C_DIS
LIN {X 33.0134,Y -14.2847,Z 60,A -31.3641,B 24.8495,C -2.83,E1 25.1453,E2 -605.5066} C_DIS
LIN {X 31.6281,Y -17.1363,Z 60,A -35.6236,B 24.8498,C -2.8272,E1 25.14,E2 -601.263} C_DIS
LIN {X 30.9871,Y -18.2699,Z 60,A -38.3292,B 24.8515,C -2.812,E1 25.1361,E2 -598.5354} C_DIS
LIN {X 29.3407,Y -20.8115,Z 60,A -42.9315,B 24.8525,C -2.8021,E1 25.1289,E2 -593.9324} C_DIS
LIN {X 27.9619,Y -22.6301,Z 60,A -46.5537,B 24.8535,C -2.7928,E1 25.1227,E2 -590.3054} C_DIS
LIN {X 26.4048,Y -24.4293,Z 60,A -50.4242,B 24.8546,C -2.7823,E1 25.1155,E2 -586.4271} C_DIS
LIN {X 24.7555,Y -26.0993,Z 60,A -54.0926,B 24.8554,C -2.7745,E1 25.1081,E2 -582.7556} C_DIS
LIN {X 22.6238,Y -27.967,Z 60,A -58.4783,B 24.8563,C -2.7664,E1 25.0988,E2 -578.3678} C_DIS
LIN {X 20.8345,Y -29.3243,Z 60,A -62.097,B 24.8571,C -2.7585,E1 25.0906,E2 -574.7434} C_DIS
LIN {X 18.8868,Y -30.6153,Z 60,A -65.6698,B 24.8576,C -2.7536,E1 25.0822,E2 -571.1704} C_DIS
LIN {X 17.1341,Y -31.6292,Z 60,A -68.7333,B 24.8579,C -2.7503,E1 25.0748,E2 -568.108} C_DIS
LIN {X 15.1495,Y -32.626,Z 60,A -72.7365,B 24.8592,C -2.7384,E1 25.0647,E2 -564.0873} C_DIS
LIN {X 13.2762,Y -33.4319,Z 60,A -75.6065,B 24.8592,C -2.7389,E1 25.0573,E2 -561.225} C_DIS
LIN {X 11.2194,Y -34.1767,Z 60,A -79.3707,B 24.8599,C -2.7309,E1 25.0473,E2 -557.4494} C_DIS
LIN {X 8.59,Y -34.9314,Z 60,A -83.1668,B 24.8596,C -2.7337,E1 25.0371,E2 -553.6659} C_DIS
LIN {X 7.3756,Y -35.2079,Z 60,A -85.6686,B 24.8605,C -2.7253,E1 25.0303,E2 -551.1473} C_DIS
LIN {X 4.4186,Y -35.6997,Z 60,A -90.3523,B 24.8607,C -2.7232,E1 25.0173,E2 -546.4629} C_DIS
LIN {X 2.028,Y -35.9147,Z 60,A -94.1716,B 24.8609,C -2.7215,E1 25.0067,E2 -542.6415} C_DIS
LIN {X 0.1425,Y -35.9633,Z 60,A -96.4694,B 24.8601,C -2.7294,E1 25.0003,E2 -540.363} C_DIS
Enddeposition()
LIN {X 0.1425,Y -35.9633,Z 60,A -96.4694,B 24.8601,C -2.7294,E1 25.0003,E2 -540.363} C_DIS
Startdeposition()
$VEL.CP = VEL_PRINT
LIN {X 0.7706,Y -35.0057,Z 60,A -94.1558,B 24.8567,C -2.7619,E1 25.007,E2 -542.7534} C_DIS
LIN {X 3.2195,Y -34.8654,Z 60,A -90.3469,B 24.8567,C -2.7612,E1 25.0176,E2 -546.5588} C_DIS
LIN {X 6.2423,Y -34.453,Z 60,A -84.6162,B 24.8554,C -2.7743,E1 25.0334,E2 -552.3149} C_DIS
LIN {X 8.9478,Y -33.8507,Z 60,A -80.7592,B 24.8559,C -2.7698,E1 25.0439,E2 -556.1556} C_DIS
LIN {X 11.3176,Y -33.1343,Z 60,A -76.8003,B 24.8555,C -2.7733,E1 25.0544,E2 -560.1155} C_DIS
LIN {X 14.119,Y -32.0413,Z 60,A -71.2656,B 24.8539,C -2.7885,E1 25.0687,E2 -565.6734} C_DIS
LIN {X 16.4212,Y -30.9246,Z 60,A -67.4638,B 24.8538,C -2.7901,E1 25.0781,E2 -569.4683} C_DIS
LIN {X 19.12,Y -29.333,Z 60,A -62.5537,B 24.8531,C -2.7965,E1 25.0898,E2 -574.3781} C_DIS
LIN {X 21.0563,Y -27.9751,Z 60,A -59.2778,B 24.8531,C -2.7959,E1 25.0972,E2 -577.6413} C_DIS
LIN {X 22.9367,Y -26.455,Z 60,A -54.364,B 24.8508,C -2.8181,E1 25.1078,E2 -582.5888} C_DIS
LIN {X 24.7225,Y -24.7951,Z 60,A -51.1044,B 24.8509,C -2.8169,E1 25.1143,E2 -585.8319} C_DIS
LIN {X 25.9045,Y -23.5566,Z 60,A -47.8058,B 24.8494,C -2.831,E1 25.1206,E2 -589.1494} C_DIS
LIN {X 27.6158,Y -21.5263,Z 60,A -43.7411,B 24.8487,C -2.8381,E1 25.1277,E2 -593.212} C_DIS
LIN {X 29.4445,Y -18.9472,Z 60,A -37.8013,B 24.8459,C -2.8635,E1 25.1371,E2 -599.1826} C_DIS
LIN {X 31.0066,Y -16.2645,Z 60,A -33.0966,B 24.845,C -2.8723,E1 25.1433,E2 -603.8835} C_DIS
LIN {X 32.4293,Y -13.2023,Z 60,A -28.057,B 24.844,C -2.8813,E1 25.149,E2 -608.9169} C_DIS
LIN {X 33.4156,Y -10.4578,Z 60,A -23.6821,B 24.8431,C -2.8898,E1 25.153,E2 -613.2873} C_DIS
LIN {X 33.7686,Y -9.255,Z 60,A -21.1706,B 24.8416,C -2.903,E1 25.1549,E2 -615.8157} C_DIS
LIN {X 34.4124,Y -6.4625,Z 60,A -16.6313,B 24.8403,C -2.9153,E1 25.1575,E2 -620.3577} C_DIS
LIN {X 34.7504,Y -4.2845,Z 60,A -12.8889,B 24.8388,C -2.9287,E1 25.1589,E2 -624.1096} C_DIS
LIN {X 34.9635,Y -1.875,Z 60,A -9.2601,B 24.838,C -2.9361,E1 25.1597,E2 -627.7345} C_DIS
LIN {X 34.9945,Y 1.1677,Z 60,A -4.0195,B 24.8358,C -2.9556,E1 25.1596,E2 -632.99} C_DIS
LIN {X 34.86,Y 3.277,Z 60,A -1.1208,B 24.8356,C -2.9579,E1 25.1589,E2 -635.8769} C_DIS
LIN {X 34.6633,Y 4.9418,Z 60,A 1.8865,B 24.8342,C -2.9703,E1 25.1578,E2 -638.8959} C_DIS
LIN {X 34.3521,Y 6.7768,Z 60,A 5.6904,B 24.8319,C -2.9909,E1 25.1558,E2 -642.7264} C_DIS
LIN {X 33.3985,Y 10.5118,Z 60,A 10.8969,B 24.8316,C -2.9931,E1 25.152,E2 -647.9082} C_DIS
LIN {X 32.657,Y 12.6287,Z 60,A 15.2693,B 24.8293,C -3.014,E1 25.1477,E2 -652.3057} C_DIS
LIN {X 31.6613,Y 14.9512,Z 60,A 19.21,B 24.8283,C -3.0225,E1 25.1432,E2 -656.2452} C_DIS
LIN {X 30.4193,Y 17.3394,Z 60,A 23.2079,B 24.8276,C -3.0283,E1 25.1379,E2 -660.2358} C_DIS
LIN {X 28.8582,Y 19.8288,Z 60,A 28.2332,B 24.8259,C -3.0435,E1 25.1302,E2 -665.2719} C_DIS
LIN {X 27.7392,Y 21.3662,Z 60,A 31.3419,B 24.825,C -3.0508,E1 25.125,E2 -668.3832} C_DIS
LIN {X 26.3826,Y 23.0203,Z 60,A 34.5308,B 24.8246,C -3.0543,E1 25.1193,E2 -671.5658} C_DIS
LIN {X 25.2653,Y 24.241,Z 60,A 37.1993,B 24.824,C -3.0596,E1 25.1142,E2 -674.2351} C_DIS
LIN {X 23.8669,Y 25.6194,Z 60,A 41.2318,B 24.822,C -3.0774,E1 25.106,E2 -678.2933} C_DIS
LIN {X 21.7758,Y 27.4187,Z 60,A 44.8059,B 24.8225,C -3.0728,E1 25.0983,E2 -681.8428} C_DIS
LIN {X 20.201,Y 28.5987,Z 60,A 48.8348,B 24.8206,C -3.0891,E1 25.0892,E2 -685.8963} C_DIS
LIN {X 18.1359,Y 29.951,Z 60,A 52.3127,B 24.8208,C -3.0876,E1 25.081,E2 -689.3595} C_DIS
LIN {X 16.4714,Y 30.8981,Z 60,A 55.637,B 24.82,C -3.0943,E1 25.0728,E2 -692.69} C_DIS
LIN {X 14.028,Y 32.0808,Z 60,A 59.9575,B 24.8196,C -3.0978,E1 25.0619,E2 -697.0077} C_DIS
LIN {X 12.3331,Y 32.7695,Z 60,A 62.587,B 24.8198,C -3.096,E1 25.0551,E2 -699.6272} C_DIS
LIN {X 10.5513,Y 33.3859,Z 60,A 66.0493,B 24.8189,C -3.1032,E1 25.0458,E2 -703.1} C_DIS
LIN {X 8.6671,Y 33.9239,Z 60,A 68.9979,B 24.8191,C -3.102,E1 25.0379,E2 -706.0411} C_DIS
LIN {X 7.1661,Y 34.273,Z 60,A 71.4524,B 24.8191,C -3.1024,E1 25.0312,E2 -708.4932} C_DIS
LIN {X 5.0128,Y 34.6532,Z 60,A 74.8173,B 24.8192,C -3.101,E1 25.022,E2 -711.8513} C_DIS
LIN {X 3.5969,Y 34.8282,Z 60,A 77.5609,B 24.8186,C -3.1062,E1 25.0143,E2 -714.6054} C_DIS
LIN {X 1.7107,Y 34.9717,Z 60,A 80.8432,B 24.8183,C -3.1084,E1 25.0052,E2 -717.8917} C_DIS
LIN {X -1.1851,Y 34.994,Z 60,A 85.0525,B 24.8192,C -3.1013,E1 24.9935,E2 -722.084} C_DIS
LIN {X -2.9538,Y 34.8884,Z 60,A 88.3291,B 24.8188,C -3.1043,E1 24.9843,E2 -725.3691} C_DIS
LIN {X -5.1802,Y 34.6278,Z 60,A 92.5383,B 24.8184,C -3.1082,E1 24.9727,E2 -729.5907} C_DIS
LIN {X -7.4683,Y 34.2079,Z 60,A 96.4282,B 24.8186,C -3.1059,E1 24.962,E2 -733.4799} C_DIS
LIN {X -11.0451,Y 33.2257,Z 60,A 101.5322,B 24.8206,C -3.0891,E1 24.9484,E2 -738.5521} C_DIS
LIN {X -12.7123,Y 32.6244,Z 60,A 104.3943,B 24.8211,C -3.085,E1 24.941,E2 -741.4104} C_DIS
LIN {X -14.1776,Y 32.0149,Z 60,A 107.2802,B 24.8211,C -3.0843,E1 24.9335,E2 -744.3014} C_DIS
LIN {X -16.2414,Y 31.0189,Z 60,A 111.5089,B 24.8213,C -3.0833,E1 24.923,E2 -748.539} C_DIS
LIN {X -18.1418,Y 29.9475,Z 60,A 114.5156,B 24.8227,C -3.0714,E1 24.9158,E2 -751.5262} C_DIS
LIN {X -19.8451,Y 28.8471,Z 60,A 118.2842,B 24.8229,C -3.0696,E1 24.907,E2 -755.3029} C_DIS
LIN {X -21.6793,Y 27.4952,Z 60,A 121.8208,B 24.824,C -3.0601,E1 24.8992,E2 -758.8296} C_DIS
LIN {X -23.6568,Y 25.8133,Z 60,A 126.5952,B 24.8245,C -3.0557,E1 24.8892,E2 -763.6125} C_DIS
LIN {X -25.4228,Y 24.0763,Z 60,A 130.0746,B 24.8262,C -3.0407,E1 24.8824,E2 -767.0708} C_DIS
LIN {X -27.0136,Y 22.2767,Z 60,A 134.5021,B 24.8268,C -3.0355,E1 24.8744,E2 -771.506} C_DIS
LIN {X -28.6106,Y 20.1838,Z 60,A 138.7755,B 24.8281,C -3.0238,E1 24.8673,E2 -775.7722} C_DIS
LIN {X -29.9696,Y 18.1054,Z 60,A 142.1196,B 24.8301,C -3.0062,E1 24.8624,E2 -779.091} C_DIS
LIN {X -30.7065,Y 16.8258,Z 60,A 145.2978,B 24.8301,C -3.0062,E1 24.858,E2 -782.2859} C_DIS
LIN {X -32.0368,Y 14.1294,Z 60,A 149.6092,B 24.8324,C -2.9864,E1 24.8529,E2 -786.5736} C_DIS
LIN {X -32.8323,Y 12.1641,Z 60,A 153.6591,B 24.833,C -2.9812,E1 24.8488,E2 -790.6337} C_DIS
LIN {X -33.4548,Y 10.3309,Z 60,A 156.2851,B 24.8346,C -2.9668,E1 24.8465,E2 -793.2403} C_DIS
LIN {X -33.9636,Y 8.5105,Z 60,A 159.9822,B 24.8351,C -2.9626,E1 24.8439,E2 -796.9488} C_DIS
LIN {X -34.4703,Y 6.1457,Z 60,A 163.9211,B 24.8364,C -2.9501,E1 24.8418,E2 -800.8811} C_DIS
LIN {X -34.7914,Y 3.9397,Z 60,A 167.1496,B 24.8381,C -2.9351,E1 24.8406,E2 -804.093} C_DIS
LIN {X -34.9546,Y 2.0315,Z 60,A 170.0524,B 24.8394,C -2.9233,E1 24.84,E2 -806.985} C_DIS
LIN {X -35.0117,Y 0.412,Z 60,A 173.0518,B 24.84,C -2.918,E1 24.8398,E2 -809.9897} C_DIS
LIN {X -34.9916,Y -1.25,Z 60,A 176.0704,B 24.8406,C -2.9122,E1 24.84,E2 -813.0125} C_DIS
LIN {X -34.8737,Y -3.1242,Z 60,A 179.1054,B 24.8417,C -2.9023,E1 24.8407,E2 -816.0422} C_DIS
LIN {X -34.6231,Y -5.2188,Z 60,A -177.4205,B 24.8429,C -2.8919,E1 24.842,E2 -819.5121} C_DIS
LIN {X -34.2806,Y -7.1288,Z 60,A -174.389,B 24.844,C -2.881,E1 24.8436,E2 -822.5355} C_DIS
LIN {X -33.9092,Y -8.725,Z 60,A -171.6806,B 24.8449,C -2.8733,E1 24.8454,E2 -825.2411} C_DIS
LIN {X -33.4354,Y -10.394,Z 60,A -168.8274,B 24.8458,C -2.8651,E1 24.8476,E2 -828.0912} C_DIS
LIN {X -32.7737,Y -12.3217,Z 60,A -165.1435,B 24.8465,C -2.8587,E1 24.8511,E2 -831.7806} C_DIS
LIN {X -31.7578,Y -14.7441,Z 60,A -161.2666,B 24.8482,C -2.8429,E1 24.8554,E2 -835.6411} C_DIS
LIN {X -31.1237,Y -16.0406,Z 60,A -158.6533,B 24.8486,C -2.8388,E1 24.8587,E2 -838.2588} C_DIS
LIN {X -30.0774,Y -17.9259,Z 60,A -155.2906,B 24.8497,C -2.8281,E1 24.8634,E2 -841.6134} C_DIS
LIN {X -29.335,Y -19.1168,Z 60,A -152.5586,B 24.8499,C -2.8264,E1 24.8675,E2 -844.3551} C_DIS
LIN {X -27.8943,Y -21.1635,Z 60,A -148.7988,B 24.8513,C -2.8134,E1 24.8737,E2 -848.102} C_DIS
LIN {X -26.5421,Y -22.8363,Z 60,A -145.075,B 24.8519,C -2.8074,E1 24.8803,E2 -851.8287} C_DIS
LIN {X -25.0244,Y -24.49,Z 60,A -141.4371,B 24.8528,C -2.7993,E1 24.8873,E2 -855.463} C_DIS
LIN {X -23.8567,Y -25.629,Z 60,A -139.0482,B 24.8537,C -2.7912,E1 24.8921,E2 -857.8425} C_DIS
LIN {X -22.3711,Y -26.9352,Z 60,A -135.1122,B 24.8536,C -2.7922,E1 24.9005,E2 -861.796} C_DIS
LIN {X -20.3942,Y -28.4615,Z 60,A -130.8431,B 24.8541,C -2.7872,E1 24.9101,E2 -866.0684} C_DIS
LIN {X -17.7502,Y -30.1813,Z 60,A -126.2351,B 24.8555,C -2.7739,E1 24.921,E2 -870.659} C_DIS
LIN {X -15.9348,Y -31.1778,Z 60,A -122.9825,B 24.8561,C -2.7681,E1 24.929,E2 -873.907} C_DIS
LIN {X -14.5082,Y -31.8664,Z 60,A -120.1264,B 24.8561,C -2.7681,E1 24.9363,E2 -876.7702} C_DIS
LIN {X -12.4432,Y -32.7282,Z 60,A -116.7238,B 24.8567,C -2.7617,E1 24.9451,E2 -880.1651} C_DIS
LIN {X -10.9635,Y -33.2527,Z 60,A -113.5541,B 24.8562,C -2.7664,E1 24.9535,E2 -883.3519} C_DIS
LIN {X -7.9233,Y -34.1055,Z 60,A -108.8936,B 24.8572,C -2.7577,E1 24.966,E2 -887.9985} C_DIS
LIN {X -5.3758,Y -34.5988,Z 60,A -104.9011,B 24.8576,C -2.7533,E1 24.977,E2 -891.9847} C_DIS
LIN {X -4.0434,Y -34.7795,Z 60,A -102.6421,B 24.8576,C -2.7536,E1 24.9833,E2 -894.2462} C_DIS
LIN {X -2.2483,Y -34.9415,Z 60,A -98.9175,B 24.8566,C -2.7629,E1 24.9937,E2 -897.9944} C_DIS
LIN {X 0.1312,Y -35.0133,Z 60,A -95.8416,B 24.8576,C -2.7537,E1 25.0022,E2 -901.0483} C_DIS
Enddeposition()
LIN {X 0.1312,Y -35.0133,Z 60,A -95.8416,B 24.8576,C -2.7537,E1 25.0022,E2 -901.0483} C_DIS
Startdeposition()
$VEL.CP = VEL_PRINT
LIN {X -0.1994,Y -34.0551,Z 60,A -98.2241,B 24.8581,C -2.7488,E1 24.9955,E2 -898.6542} C_DIS
Enddeposition()
END
